KUKA KRL program: EPS_2_25618_SANMH10_A_20250918115518.src

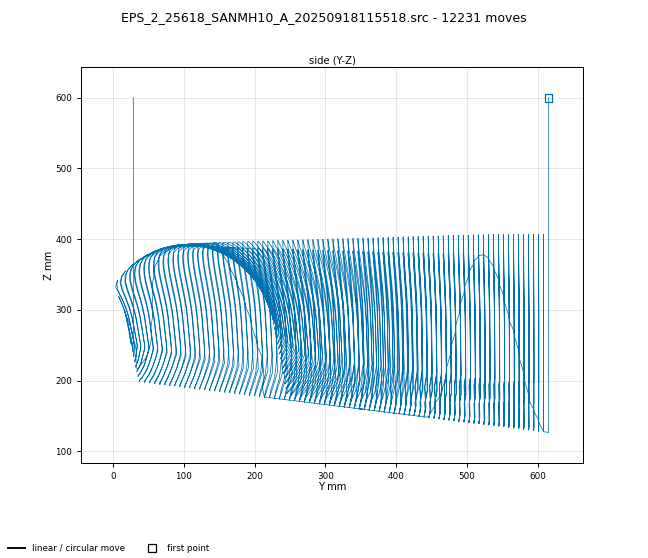
[picture p0: tool path of EPS_2_25618_SANMH10_A_20250918115518.src, 12231 of 12233 moves have a stored position in this frame; points joined in program order, loops and branches not executed]
&ACCESS RVP
&REL 4
&COMMENT QRS 19112012
&PARAM EDITMASK = *
DEF PART()
EXT BAS (BAS_COMMAND :IN,REAL :IN )
INT I
BAS (#INITMOV,0 )

;KUKA QRS Post kuka4.cps  Date:22-06-2017 !

File_ID=2846

QRS_PRE_INIT()

;Init var - Until changes are made in qrs_pre_init
Outlet_Square_prg=0
Inlet_1_Square_prg=0
Inlet_2_Square_prg=0
Inlet_3_Square_prg=0
Inlet_4_Square_prg=0
Inlet_5_Square_prg=0

Outlet_1={X 0.000, Y 546.330, Z 306.500, B 0.000, E1 0.000 }
Inlet_1={X 0.000, Y 548.460, Z 276.500, B 0.000, E1 118.000 }
Outlet_1_type=201
Inlet_1_type=201
;QRS#1=Sidecore dimensions
;QRS#2=200-8" PVC SDR 35
;QRS#3=200-8" PVC SDR 35
;QRS#4=
;QRS#5=
;QRS#6=
;QRS#7=
;QRS#8=
;QRS#9=12-08 PSX
;QRS#10=12-08 PSX
;QRS#11=
;QRS#12=
;QRS#13=
;QRS#14=
;QRS#15=
;QRS#16=1220x127x686 2,25'
;QRS#17=EPS Height
;QRS#18=407
;QRS#19=*
;QRS#20= UPDATED VERSION 22-06-2017
;QRS#21=*
Outlet_Square=0100
Inlet_1_Square=0100
Inlet_2_Square=0
Inlet_3_Square=0
Inlet_4_Square=0
Inlet_5_Square=0
Mill_Square=1
Outlet_Square_Prg=204
Inlet_1_Square_prg=204

QRS_INIT()

$ADVANCE=5

; T1
PTP {E1 173.646,E2 173.646}
PTP {X 0,Y 615.451,A -85,B 0,C 180,E1 173.646,E2 173.646,E3 0,E4 0,E5 0,E6 0}
QRS_SPEED_INIT()
LIN {X 0,Y 615.451,Z 600,A -85,B 0,C 180,E1 173.646,E2 173.646,E3 0,E4 0,E5 0,E6 0} C_VEL
LIN {X 0,Y 615.451,Z 136.872,A -85,B 0,C 180,E1 173.646,E2 173.646} C_VEL
LIN {X 0,Y 615.451,Z 128.693,A -85,B 0,C 180,E1 173.646,E2 173.646} C_VEL
LIN {X 0,Y 615.444,Z 126.693,A -85,B 0,C 180,E1 173.46,E2 173.46} C_VEL
LIN {X 0,Y 615.447,Z 126.714,A -85,B 0,C 180,E1 171.214,E2 171.214} C_VEL
LIN {X 0,Y 615.498,Z 142.353,A -85,B 0,C 180,E1 168.64,E2 168.64} C_VEL
LIN {X 0,Y 615.49,Z 160.105,A -85,B 0,C 180,E1 165.759,E2 165.759} C_VEL
LIN {X 0,Y 615.486,Z 165.964,A -85,B 0,C 180,E1 164.816,E2 164.816} C_VEL
LIN {X 0,Y 615.488,Z 273.613,A -85,B 0,C 180,E1 163.53,E2 163.53} C_VEL
LIN {X 0,Y 615.478,Z 286.482,A -85,B 0,C 180,E1 163.242,E2 163.242} C_VEL
LIN {X 0,Y 615.49,Z 299.343,A -85,B 0,C 180,E1 162.815,E2 162.815} C_VEL
LIN {X 0,Y 615.492,Z 310.759,A -85,B 0,C 180,E1 162.301,E2 162.301} C_VEL
LIN {X 0,Y 615.481,Z 322.204,A -85,B 0,C 180,E1 161.638,E2 161.638} C_VEL
LIN {X 0,Y 615.499,Z 333.228,A -85,B 0,C 180,E1 160.835,E2 160.835} C_VEL
LIN {X 0,Y 615.498,Z 342.752,A -85,B 0,C 180,E1 159.967,E2 159.967} C_VEL
LIN {X 0,Y 615.498,Z 350.589,A -85,B 0,C 180,E1 159.094,E2 159.094} C_VEL
LIN {X 0,Y 615.498,Z 358.274,A -85,B 0,C 180,E1 158.04,E2 158.04} C_VEL
LIN {X 0,Y 615.497,Z 363.428,A -85,B 0,C 180,E1 157.156,E2 157.156} C_VEL
LIN {X 0,Y 615.495,Z 368.74,A -85,B 0,C 180,E1 155.991,E2 155.991} C_VEL
LIN {X 0,Y 615.496,Z 372.068,A -85,B 0,C 180,E1 155.008,E2 155.008} C_VEL
LIN {X 0,Y 615.493,Z 373.871,A -85,B 0,C 180,E1 154.284,E2 154.284} C_VEL
LIN {X 0,Y 615.498,Z 375.211,A -85,B 0,C 180,E1 153.556,E2 153.556} C_VEL
LIN {X 0,Y 615.493,Z 376.024,A -85,B 0,C 180,E1 152.823,E2 152.823} C_VEL
LIN {X 0,Y 615.498,Z 376.298,A -85,B 0,C 180,E1 151.549,E2 151.549} C_VEL
LIN {X 0,Y 615.497,Z 374.962,A -85,B 0,C 180,E1 150.205,E2 150.205} C_VEL
LIN {X 0,Y 615.495,Z 372.101,A -85,B 0,C 180,E1 148.914,E2 148.914} C_VEL
LIN {X 0,Y 615.494,Z 369.013,A -85,B 0,C 180,E1 147.992,E2 147.992} C_VEL
LIN {X 0,Y 615.496,Z 363.479,A -85,B 0,C 180,E1 146.764,E2 146.764} C_VEL
LIN {X 0,Y 615.496,Z 356.718,A -85,B 0,C 180,E1 145.639,E2 145.639} C_VEL
LIN {X 0,Y 615.495,Z 348.697,A -85,B 0,C 180,E1 144.585,E2 144.585} C_VEL
LIN {X 0,Y 615.495,Z 340.536,A -85,B 0,C 180,E1 143.723,E2 143.723} C_VEL
LIN {X 0,Y 615.498,Z 331.142,A -85,B 0,C 180,E1 142.911,E2 142.911} C_VEL
LIN {X 0,Y 615.464,Z 320.86,A -85,B 0,C 180,E1 142.184,E2 142.184} C_VEL
LIN {X 0,Y 615.468,Z 309.903,A -85,B 0,C 180,E1 141.565,E2 141.565} C_VEL
LIN {X 0,Y 615.497,Z 297.229,A -85,B 0,C 180,E1 141.017,E2 141.017} C_VEL
LIN {X 0,Y 615.49,Z 285.344,A -85,B 0,C 180,E1 140.637,E2 140.637} C_VEL
LIN {X 0,Y 615.494,Z 272.35,A -85,B 0,C 180,E1 140.358,E2 140.358} C_VEL
LIN {X 0,Y 615.497,Z 165.933,A -85,B 0,C 180,E1 139.09,E2 139.09} C_VEL
LIN {X 0,Y 615.494,Z 148.019,A -85,B 0,C 180,E1 136.193,E2 136.193} C_VEL
LIN {X 0,Y 615.499,Z 130.019,A -85,B 0,C 180,E1 133.244,E2 133.244} C_VEL
LIN {X 0,Y 615.452,Z 126.693,A -85,B 0,C 180,E1 132.659,E2 132.659} C_VEL
LIN {X 0,Y 615.434,Z 126.696,A -85,B 0,C 180,E1 130.082,E2 130.082} C_VEL
LIN {X 0,Y 615.438,Z 126.697,A -85,B 0,C 180,E1 128.005,E2 128.005} C_VEL
LIN {X 0,Y 615.477,Z 126.699,A -85,B 0,C 180,E1 125.617,E2 125.617} C_VEL
LIN {X 0,Y 615.485,Z 126.694,A -85,B 0,C 180,E1 123.237,E2 123.237} C_VEL
LIN {X 0,Y 615.452,Z 126.693,A -85,B 0,C 180,E1 120.922,E2 120.922} C_VEL
LIN {X 0,Y 615.431,Z 126.696,A -85,B 0,C 180,E1 118.44,E2 118.44} C_VEL
LIN {X 0,Y 615.498,Z 126.697,A -85,B 0,C 180,E1 115.57,E2 115.57} C_VEL
LIN {X 0,Y 615.435,Z 126.695,A -85,B 0,C 180,E1 112.847,E2 112.847} C_VEL
LIN {X 0,Y 615.431,Z 126.697,A -85,B 0,C 180,E1 110.541,E2 110.541} C_VEL
LIN {X 0,Y 615.48,Z 126.699,A -85,B 0,C 180,E1 107.958,E2 107.958} C_VEL
LIN {X 0,Y 615.448,Z 126.694,A -85,B 0,C 180,E1 105.228,E2 105.228} C_VEL
LIN {X 0,Y 615.443,Z 126.694,A -85,B 0,C 180,E1 103.203,E2 103.203} C_VEL
LIN {X 0,Y 615.428,Z 126.696,A -85,B 0,C 180,E1 100.857,E2 100.857} C_VEL
LIN {X 0,Y 615.439,Z 126.698,A -85,B 0,C 180,E1 98.538,E2 98.538} C_VEL
LIN {X 0,Y 615.499,Z 126.694,A -85,B 0,C 180,E1 95.899,E2 95.899} C_VEL
LIN {X 0,Y 615.433,Z 126.695,A -85,B 0,C 180,E1 93.274,E2 93.274} C_VEL
LIN {X 0,Y 615.432,Z 126.696,A -85,B 0,C 180,E1 91.309,E2 91.309} C_VEL
LIN {X 0,Y 615.432,Z 126.696,A -85,B 0,C 180,E1 89.346,E2 89.346} C_VEL
LIN {X 0,Y 615.432,Z 126.696,A -85,B 0,C 180,E1 87.382,E2 87.382} C_VEL
LIN {X 0,Y 615.431,Z 126.696,A -85,B 0,C 180,E1 85.416,E2 85.416} C_VEL
LIN {X 0,Y 615.43,Z 126.696,A -85,B 0,C 180,E1 83.443,E2 83.443} C_VEL
LIN {X 0,Y 615.429,Z 126.696,A -85,B 0,C 180,E1 81.463,E2 81.463} C_VEL
LIN {X 0,Y 615.429,Z 126.697,A -85,B 0,C 180,E1 79.143,E2 79.143} C_VEL
LIN {X 0,Y 615.454,Z 126.699,A -85,B 0,C 180,E1 76.799,E2 76.799} C_VEL
LIN {X 0,Y 615.464,Z 126.695,A -85,B 0,C 180,E1 74.095,E2 74.095} C_VEL
LIN {X 0,Y 615.425,Z 126.697,A -85,B 0,C 180,E1 71.414,E2 71.414} C_VEL
LIN {X 0,Y 615.497,Z 126.698,A -85,B 0,C 180,E1 68.569,E2 68.569} C_VEL
LIN {X 0,Y 615.425,Z 126.697,A -85,B 0,C 180,E1 65.726,E2 65.726} C_VEL
LIN {X 0,Y 615.425,Z 126.697,A -85,B 0,C 180,E1 63.554,E2 63.554} C_VEL
LIN {X 0,Y 615.482,Z 126.697,A -85,B 0,C 180,E1 60.594,E2 60.594} C_VEL
LIN {X 0,Y 615.449,Z 126.696,A -85,B 0,C 180,E1 58.313,E2 58.313} C_VEL
LIN {X 0,Y 615.425,Z 126.697,A -85,B 0,C 180,E1 55.975,E2 55.975} C_VEL
LIN {X 0,Y 615.484,Z 126.7,A -85,B 0,C 180,E1 53.065,E2 53.065} C_VEL
LIN {X 0,Y 615.428,Z 126.697,A -85,B 0,C 180,E1 50.246,E2 50.246} C_VEL
LIN {X 0,Y 615.421,Z 126.698,A -85,B 0,C 180,E1 47.927,E2 47.927} C_VEL
LIN {X 0,Y 615.425,Z 126.698,A -85,B 0,C 180,E1 45.846,E2 45.846} C_VEL
LIN {X 0,Y 615.487,Z 126.7,A -85,B 0,C 180,E1 43.245,E2 43.245} C_VEL
LIN {X 0,Y 615.44,Z 126.697,A -85,B 0,C 180,E1 40.611,E2 40.611} C_VEL
LIN {X 0,Y 615.467,Z 126.696,A -85,B 0,C 180,E1 38.906,E2 38.906} C_VEL
LIN {X 0,Y 615.424,Z 126.697,A -85,B 0,C 180,E1 36.43,E2 36.43} C_VEL
LIN {X 0,Y 615.471,Z 126.701,A -85,B 0,C 180,E1 33.533,E2 33.533} C_VEL
LIN {X 0,Y 615.448,Z 126.697,A -85,B 0,C 180,E1 30.922,E2 30.922} C_VEL
LIN {X 0,Y 615.42,Z 126.698,A -85,B 0,C 180,E1 28.44,E2 28.44} C_VEL
LIN {X 0,Y 615.471,Z 126.7,A -85,B 0,C 180,E1 25.717,E2 25.717} C_VEL
LIN {X 0,Y 615.428,Z 126.698,A -85,B 0,C 180,E1 22.847,E2 22.847} C_VEL
LIN {X 0,Y 615.419,Z 126.698,A -85,B 0,C 180,E1 20.542,E2 20.542} C_VEL
LIN {X 0,Y 615.461,Z 126.7,A -85,B 0,C 180,E1 17.958,E2 17.958} C_VEL
LIN {X 0,Y 615.443,Z 126.698,A -85,B 0,C 180,E1 15.227,E2 15.227} C_VEL
LIN {X 0,Y 615.437,Z 126.698,A -85,B 0,C 180,E1 13.203,E2 13.203} C_VEL
LIN {X 0,Y 615.417,Z 126.699,A -85,B 0,C 180,E1 10.858,E2 10.858} C_VEL
LIN {X 0,Y 615.426,Z 126.699,A -85,B 0,C 180,E1 8.538,E2 8.538} C_VEL
LIN {X 0,Y 615.498,Z 126.699,A -85,B 0,C 180,E1 5.899,E2 5.899} C_VEL
LIN {X 0,Y 615.425,Z 126.698,A -85,B 0,C 180,E1 3.273,E2 3.273} C_VEL
LIN {X 0,Y 615.424,Z 126.699,A -85,B 0,C 180,E1 1.309,E2 1.309} C_VEL
LIN {X 0,Y 615.424,Z 126.698,A -85,B 0,C 180,E1 -0.654,E2 -0.654} C_VEL
LIN {X 0,Y 615.424,Z 126.699,A -85,B 0,C 180,E1 -2.618,E2 -2.618} C_VEL
LIN {X 0,Y 615.423,Z 126.699,A -85,B 0,C 180,E1 -4.585,E2 -4.585} C_VEL
LIN {X 0,Y 615.422,Z 126.699,A -85,B 0,C 180,E1 -6.557,E2 -6.557} C_VEL
LIN {X 0,Y 615.421,Z 126.699,A -85,B 0,C 180,E1 -8.537,E2 -8.537} C_VEL
LIN {X 0,Y 615.416,Z 126.699,A -85,B 0,C 180,E1 -10.858,E2 -10.858} C_VEL
LIN {X 0,Y 615.438,Z 126.7,A -85,B 0,C 180,E1 -13.202,E2 -13.202} C_VEL
LIN {X 0,Y 615.461,Z 126.699,A -85,B 0,C 180,E1 -15.906,E2 -15.906} C_VEL
LIN {X 0,Y 615.414,Z 126.7,A -85,B 0,C 180,E1 -18.648,E2 -18.648} C_VEL
LIN {X 0,Y 615.49,Z 126.7,A -85,B 0,C 180,E1 -21.432,E2 -21.432} C_VEL
LIN {X 0,Y 615.416,Z 126.699,A -85,B 0,C 180,E1 -24.275,E2 -24.275} C_VEL
LIN {X 0,Y 615.413,Z 126.7,A -85,B 0,C 180,E1 -26.448,E2 -26.448} C_VEL
LIN {X 0,Y 615.477,Z 126.702,A -85,B 0,C 180,E1 -29.407,E2 -29.407} C_VEL
LIN {X 0,Y 615.445,Z 126.7,A -85,B 0,C 180,E1 -31.688,E2 -31.688} C_VEL
LIN {X 0,Y 615.416,Z 126.7,A -85,B 0,C 180,E1 -34.027,E2 -34.027} C_VEL
LIN {X 0,Y 615.463,Z 126.7,A -85,B 0,C 180,E1 -36.935,E2 -36.935} C_VEL
LIN {X 0,Y 615.423,Z 126.7,A -85,B 0,C 180,E1 -39.755,E2 -39.755} C_VEL
LIN {X 0,Y 615.411,Z 126.7,A -85,B 0,C 180,E1 -42.073,E2 -42.073} C_VEL
LIN {X 0,Y 615.413,Z 126.7,A -85,B 0,C 180,E1 -44.156,E2 -44.156} C_VEL
LIN {X 0,Y 615.412,Z 126.7,A -85,B 0,C 180,E1 -46.01,E2 -46.01} C_VEL
LIN {X 0,Y 615.444,Z 126.7,A -85,B 0,C 180,E1 -48.524,E2 -48.524} C_VEL
LIN {X 0,Y 615.466,Z 126.7,A -85,B 0,C 180,E1 -51.095,E2 -51.095} C_VEL
LIN {X 0,Y 615.417,Z 126.7,A -85,B 0,C 180,E1 -53.571,E2 -53.571} C_VEL
LIN {X 0,Y 615.459,Z 126.699,A -85,B 0,C 180,E1 -56.47,E2 -56.47} C_VEL
LIN {X 0,Y 615.448,Z 126.7,A -85,B 0,C 180,E1 -59.079,E2 -59.079} C_VEL
LIN {X 0,Y 615.414,Z 126.699,A -85,B 0,C 180,E1 -61.563,E2 -61.563} C_VEL
LIN {X 0,Y 615.414,Z 126.699,A -85,B 0,C 180,E1 -63.553,E2 -63.553} C_VEL
LIN {X 0,Y 615.433,Z 126.699,A -85,B 0,C 180,E1 -66.004,E2 -66.004} C_VEL
LIN {X 0,Y 615.424,Z 126.78,A -85,B 0,C 180,E1 -67.838,E2 -67.838} C_VEL
LIN {X 0,Y 615.496,Z 145.823,A -85,B 0,C 180,E1 -70.49,E2 -70.49} C_VEL
LIN {X 0,Y 615.458,Z 165.936,A -85,B 0,C 180,E1 -73.242,E2 -73.242} C_VEL
LIN {X 0,Y 615.475,Z 185.711,A -85,B 0,C 180,E1 -75.916,E2 -75.916} C_VEL
LIN {X 0,Y 615.46,Z 194.649,A -85,B 0,C 180,E1 -77.114,E2 -77.114} C_VEL
LIN {X 0,Y 615.488,Z 302.864,A -85,B 0,C 180,E1 -78.411,E2 -78.411} C_VEL
LIN {X 0,Y 615.477,Z 315.368,A -85,B 0,C 180,E1 -78.682,E2 -78.682} C_VEL
LIN {X 0,Y 615.488,Z 328.616,A -85,B 0,C 180,E1 -79.113,E2 -79.113} C_VEL
LIN {X 0,Y 615.477,Z 340.49,A -85,B 0,C 180,E1 -79.64,E2 -79.64} C_VEL
LIN {X 0,Y 615.494,Z 352.003,A -85,B 0,C 180,E1 -80.305,E2 -80.305} C_VEL
LIN {X 0,Y 615.499,Z 362.349,A -85,B 0,C 180,E1 -81.05,E2 -81.05} C_VEL
LIN {X 0,Y 615.497,Z 370.818,A -85,B 0,C 180,E1 -81.795,E2 -81.795} C_VEL
LIN {X 0,Y 615.498,Z 378.611,A -85,B 0,C 180,E1 -82.62,E2 -82.62} C_VEL
LIN {X 0,Y 615.496,Z 386.207,A -85,B 0,C 180,E1 -83.609,E2 -83.609} C_VEL
LIN {X 0,Y 615.498,Z 393.208,A -85,B 0,C 180,E1 -84.759,E2 -84.759} C_VEL
LIN {X 0,Y 615.494,Z 397.854,A -85,B 0,C 180,E1 -85.744,E2 -85.744} C_VEL
LIN {X 0,Y 615.494,Z 401.401,A -85,B 0,C 180,E1 -86.728,E2 -86.728} C_VEL
LIN {X 0,Y 615.497,Z 403.234,A -85,B 0,C 180,E1 -87.383,E2 -87.383} C_VEL
LIN {X 0,Y 615.5,Z 404.608,A -85,B 0,C 180,E1 -88.038,E2 -88.038} C_VEL
LIN {X 0,Y 615.496,Z 406.174,A -85,B 0,C 180,E1 -89.346,E2 -89.346} C_VEL
LIN {X 0,Y 615.494,Z 406.389,A -85,B 0,C 180,E1 -90.001,E2 -90.001} C_VEL
LIN {X 0,Y 615.495,Z 405.579,A -85,B 0,C 180,E1 -91.309,E2 -91.309} C_VEL
LIN {X 0,Y 615.5,Z 404.607,A -85,B 0,C 180,E1 -91.964,E2 -91.964} C_VEL
LIN {X 0,Y 615.497,Z 403.232,A -85,B 0,C 180,E1 -92.618,E2 -92.618} C_VEL
LIN {X 0,Y 615.496,Z 400.348,A -85,B 0,C 180,E1 -93.601,E2 -93.601} C_VEL
LIN {X 0,Y 615.498,Z 396.439,A -85,B 0,C 180,E1 -94.585,E2 -94.585} C_VEL
LIN {X 0,Y 615.499,Z 391.402,A -85,B 0,C 180,E1 -95.57,E2 -95.57} C_VEL
LIN {X 0,Y 615.497,Z 384.869,A -85,B 0,C 180,E1 -96.583,E2 -96.583} C_VEL
LIN {X 0,Y 615.497,Z 377.128,A -85,B 0,C 180,E1 -97.546,E2 -97.546} C_VEL
LIN {X 0,Y 615.498,Z 369.039,A -85,B 0,C 180,E1 -98.372,E2 -98.372} C_VEL
LIN {X 0,Y 615.499,Z 359.16,A -85,B 0,C 180,E1 -99.199,E2 -99.199} C_VEL
LIN {X 0,Y 615.488,Z 347.972,A -85,B 0,C 180,E1 -99.946,E2 -99.946} C_VEL
LIN {X 0,Y 615.482,Z 337.012,A -85,B 0,C 180,E1 -100.528,E2 -100.528} C_VEL
LIN {X 0,Y 615.48,Z 324.482,A -85,B 0,C 180,E1 -101.04,E2 -101.04} C_VEL
LIN {X 0,Y 615.479,Z 312.044,A -85,B 0,C 180,E1 -101.402,E2 -101.402} C_VEL
LIN {X 0,Y 615.493,Z 298.427,A -85,B 0,C 180,E1 -101.652,E2 -101.652} C_VEL
LIN {X 0,Y 615.46,Z 194.641,A -85,B 0,C 180,E1 -102.888,E2 -102.888} C_VEL
LIN {X 0,Y 615.497,Z 173.46,A -85,B 0,C 180,E1 -105.735,E2 -105.735} C_VEL
LIN {X 0,Y 615.482,Z 152.104,A -85,B 0,C 180,E1 -108.647,E2 -108.647} C_VEL
LIN {X 0,Y 615.494,Z 131.977,A -85,B 0,C 180,E1 -111.432,E2 -111.432} C_VEL
LIN {X 0,Y 615.423,Z 126.699,A -85,B 0,C 180,E1 -112.187,E2 -112.187} C_VEL
LIN {X 0,Y 615.418,Z 126.699,A -85,B 0,C 180,E1 -114.275,E2 -114.275} C_VEL
LIN {X 0,Y 615.418,Z 126.699,A -85,B 0,C 180,E1 -116.448,E2 -116.448} C_VEL
LIN {X 0,Y 615.479,Z 126.7,A -85,B 0,C 180,E1 -119.407,E2 -119.407} C_VEL
LIN {X 0,Y 615.448,Z 126.697,A -85,B 0,C 180,E1 -121.688,E2 -121.688} C_VEL
LIN {X 0,Y 615.422,Z 126.698,A -85,B 0,C 180,E1 -124.027,E2 -124.027} C_VEL
LIN {X 0,Y 615.48,Z 126.7,A -85,B 0,C 180,E1 -126.935,E2 -126.935} C_VEL
LIN {X 0,Y 615.428,Z 126.697,A -85,B 0,C 180,E1 -129.755,E2 -129.755} C_VEL
LIN {X 0,Y 615.424,Z 126.698,A -85,B 0,C 180,E1 -132.073,E2 -132.073} C_VEL
LIN {X 0,Y 615.428,Z 126.698,A -85,B 0,C 180,E1 -134.155,E2 -134.155} C_VEL
LIN {X 0,Y 615.493,Z 126.7,A -85,B 0,C 180,E1 -136.756,E2 -136.756} C_VEL
LIN {X 0,Y 615.442,Z 126.695,A -85,B 0,C 180,E1 -139.39,E2 -139.39} C_VEL
LIN {X 0,Y 615.43,Z 126.697,A -85,B 0,C 180,E1 -141.927,E2 -141.927} C_VEL
LIN {X 0,Y 615.47,Z 126.699,A -85,B 0,C 180,E1 -144.383,E2 -144.383} C_VEL
LIN {X 0,Y 615.485,Z 126.695,A -85,B 0,C 180,E1 -146.764,E2 -146.764} C_VEL
LIN {X 0,Y 615.452,Z 126.694,A -85,B 0,C 180,E1 -149.078,E2 -149.078} C_VEL
LIN {X 0,Y 615.431,Z 126.696,A -85,B 0,C 180,E1 -151.56,E2 -151.56} C_VEL
LIN {X 0,Y 615.498,Z 126.697,A -85,B 0,C 180,E1 -154.43,E2 -154.43} C_VEL
LIN {X 0,Y 615.437,Z 126.695,A -85,B 0,C 180,E1 -157.153,E2 -157.153} C_VEL
LIN {X 0,Y 615.435,Z 126.696,A -85,B 0,C 180,E1 -159.457,E2 -159.457} C_VEL
LIN {X 0,Y 615.489,Z 126.7,A -85,B 0,C 180,E1 -162.043,E2 -162.043} C_VEL
LIN {X 0,Y 615.451,Z 126.693,A -85,B 0,C 180,E1 -164.773,E2 -164.773} C_VEL
LIN {X 0,Y 615.447,Z 126.693,A -85,B 0,C 180,E1 -166.798,E2 -166.798} C_VEL
LIN {X 0,Y 615.437,Z 126.695,A -85,B 0,C 180,E1 -169.138,E2 -169.138} C_VEL
LIN {X 0,Y 615.455,Z 126.697,A -85,B 0,C 180,E1 -171.463,E2 -171.463} C_VEL
LIN {X 0,Y 615.499,Z 126.69,A -85,B 0,C 180,E1 -174.102,E2 -174.102} C_VEL
LIN {X 0,Y 615.442,Z 126.693,A -85,B 0,C 180,E1 -176.727,E2 -176.727} C_VEL
LIN {X 0,Y 615.442,Z 126.693,A -85,B 0,C 180,E1 -178.691,E2 -178.691} C_VEL
LIN {X 0,Y 615.466,Z 126.698,A -85,B 0,C 180,E1 -181.309,E2 -181.309} C_VEL
LIN {X 0,Y 615.486,Z 126.691,A -85,B 0,C 180,E1 -183.929,E2 -183.929} C_VEL
LIN {X 0,Y 615.444,Z 126.693,A -85,B 0,C 180,E1 -186.54,E2 -186.54} C_VEL
LIN {X 0,Y 614.772,Z 126.843,A -85,B 0,C 180,E1 -186.904,E2 -186.904} C_VEL
LIN {X 0,Y 611.949,Z 127.262,A -85,B 0,C 180,E1 -187.474,E2 -187.474} C_VEL
LIN {X 0,Y 609.112,Z 127.617,A -85,B 0,C 180,E1 -188.048,E2 -188.048} C_VEL
LIN {X 0,Y 608.43,Z 127.691,A -85,B 0,C 180,E1 -188.418,E2 -188.418} C_VEL
LIN {X 0,Y 608.425,Z 127.751,A -85,B 0,C 180,E1 -188.72,E2 -188.72} C_VEL
LIN {X 0,Y 608.481,Z 141.815,A -85,B 0,C 180,E1 -191.058,E2 -191.058} C_VEL
LIN {X 0,Y 608.474,Z 159.127,A -85,B 0,C 180,E1 -193.894,E2 -193.894} C_VEL
LIN {X 0,Y 608.461,Z 166.295,A -85,B 0,C 180,E1 -195.042,E2 -195.042} C_VEL
LIN {X 0,Y 608.556,Z 273.083,A -85,B 0,C 180,E1 -196.324,E2 -196.324} C_VEL
LIN {X 0,Y 608.524,Z 286.825,A -85,B 0,C 180,E1 -196.633,E2 -196.633} C_VEL
LIN {X 0,Y 608.524,Z 298.998,A -85,B 0,C 180,E1 -197.042,E2 -197.042} C_VEL
LIN {X 0,Y 608.52,Z 310.581,A -85,B 0,C 180,E1 -197.562,E2 -197.562} C_VEL
LIN {X 0,Y 608.478,Z 322.455,A -85,B 0,C 180,E1 -198.253,E2 -198.253} C_VEL
LIN {X 0,Y 608.471,Z 333.275,A -85,B 0,C 180,E1 -199.044,E2 -199.044} C_VEL
LIN {X 0,Y 608.467,Z 342.896,A -85,B 0,C 180,E1 -199.922,E2 -199.922} C_VEL
LIN {X 0,Y 608.456,Z 350.516,A -85,B 0,C 180,E1 -200.768,E2 -200.768} C_VEL
LIN {X 0,Y 608.456,Z 358.581,A -85,B 0,C 180,E1 -201.87,E2 -201.87} C_VEL
LIN {X 0,Y 608.447,Z 363.797,A -85,B 0,C 180,E1 -202.765,E2 -202.765} C_VEL
LIN {X 0,Y 608.441,Z 368.826,A -85,B 0,C 180,E1 -203.846,E2 -203.846} C_VEL
LIN {X 0,Y 608.433,Z 372.58,A -85,B 0,C 180,E1 -204.937,E2 -204.937} C_VEL
LIN {X 0,Y 608.427,Z 375.165,A -85,B 0,C 180,E1 -206.037,E2 -206.037} C_VEL
LIN {X 0,Y 608.435,Z 376.654,A -85,B 0,C 180,E1 -207.198,E2 -207.198} C_VEL
LIN {X 0,Y 608.423,Z 376.851,A -85,B 0,C 180,E1 -208.611,E2 -208.611} C_VEL
LIN {X 0,Y 608.422,Z 375.314,A -85,B 0,C 180,E1 -209.963,E2 -209.963} C_VEL
LIN {X 0,Y 608.442,Z 374.141,A -85,B 0,C 180,E1 -210.547,E2 -210.547} C_VEL
LIN {X 0,Y 608.429,Z 370.828,A -85,B 0,C 180,E1 -211.707,E2 -211.707} C_VEL
LIN {X 0,Y 608.447,Z 366.018,A -85,B 0,C 180,E1 -212.881,E2 -212.881} C_VEL
LIN {X 0,Y 608.441,Z 359.505,A -85,B 0,C 180,E1 -214.072,E2 -214.072} C_VEL
LIN {X 0,Y 608.467,Z 352.616,A -85,B 0,C 180,E1 -215.062,E2 -215.062} C_VEL
LIN {X 0,Y 608.46,Z 343.639,A -85,B 0,C 180,E1 -216.092,E2 -216.092} C_VEL
LIN {X 0,Y 608.492,Z 333.766,A -85,B 0,C 180,E1 -217.005,E2 -217.005} C_VEL
LIN {X 0,Y 608.463,Z 323.824,A -85,B 0,C 180,E1 -217.747,E2 -217.747} C_VEL
LIN {X 0,Y 608.471,Z 313.346,A -85,B 0,C 180,E1 -218.381,E2 -218.381} C_VEL
LIN {X 0,Y 608.506,Z 301.271,A -85,B 0,C 180,E1 -218.957,E2 -218.957} C_VEL
LIN {X 0,Y 608.551,Z 288.756,A -85,B 0,C 180,E1 -219.402,E2 -219.402} C_VEL
LIN {X 0,Y 608.537,Z 275.769,A -85,B 0,C 180,E1 -219.717,E2 -219.717} C_VEL
LIN {X 0,Y 608.552,Z 255.918,A -85,B 0,C 180,E1 -219.985,E2 -219.985} C_VEL
LIN {X 0,Y 608.47,Z 166.173,A -85,B 0,C 180,E1 -221.053,E2 -221.053} C_VEL
LIN {X 0,Y 608.478,Z 148.886,A -85,B 0,C 180,E1 -223.869,E2 -223.869} C_VEL
LIN {X 0,Y 608.507,Z 131.819,A -85,B 0,C 180,E1 -226.688,E2 -226.688} C_VEL
LIN {X 0,Y 608.437,Z 127.691,A -85,B 0,C 180,E1 -227.386,E2 -227.386} C_VEL
LIN {X 0,Y 608.422,Z 127.691,A -85,B 0,C 180,E1 -229.694,E2 -229.694} C_VEL
LIN {X 0,Y 608.444,Z 127.693,A -85,B 0,C 180,E1 -232.251,E2 -232.251} C_VEL
LIN {X 0,Y 608.42,Z 127.694,A -85,B 0,C 180,E1 -235.099,E2 -235.099} C_VEL
LIN {X 0,Y 608.417,Z 127.692,A -85,B 0,C 180,E1 -237.485,E2 -237.485} C_VEL
LIN {X 0,Y 608.454,Z 127.694,A -85,B 0,C 180,E1 -240.219,E2 -240.219} C_VEL
LIN {X 0,Y 608.406,Z 127.693,A -85,B 0,C 180,E1 -243.223,E2 -243.223} C_VEL
LIN {X 0,Y 608.417,Z 127.692,A -85,B 0,C 180,E1 -245.427,E2 -245.427} C_VEL
LIN {X 0,Y 608.457,Z 127.697,A -85,B 0,C 180,E1 -248.308,E2 -248.308} C_VEL
LIN {X 0,Y 608.418,Z 127.692,A -85,B 0,C 180,E1 -251.3,E2 -251.3} C_VEL
LIN {X 0,Y 608.442,Z 127.695,A -85,B 0,C 180,E1 -253.905,E2 -253.905} C_VEL
LIN {X 0,Y 608.436,Z 127.692,A -85,B 0,C 180,E1 -256.642,E2 -256.642} C_VEL
LIN {X 0,Y 608.417,Z 127.693,A -85,B 0,C 180,E1 -259.349,E2 -259.349} C_VEL
LIN {X 0,Y 608.476,Z 127.694,A -85,B 0,C 180,E1 -262.033,E2 -262.033} C_VEL
LIN {X 0,Y 608.421,Z 127.692,A -85,B 0,C 180,E1 -264.697,E2 -264.697} C_VEL
LIN {X 0,Y 608.438,Z 127.692,A -85,B 0,C 180,E1 -267.351,E2 -267.351} C_VEL
LIN {X 0,Y 608.478,Z 127.692,A -85,B 0,C 180,E1 -269.999,E2 -269.999} C_VEL
LIN {X 0,Y 608.428,Z 127.691,A -85,B 0,C 180,E1 -272.648,E2 -272.648} C_VEL
LIN {X 0,Y 608.431,Z 127.694,A -85,B 0,C 180,E1 -275.302,E2 -275.302} C_VEL
LIN {X 0,Y 608.469,Z 127.69,A -85,B 0,C 180,E1 -277.966,E2 -277.966} C_VEL
LIN {X 0,Y 608.41,Z 127.693,A -85,B 0,C 180,E1 -280.65,E2 -280.65} C_VEL
LIN {X 0,Y 608.438,Z 127.697,A -85,B 0,C 180,E1 -283.356,E2 -283.356} C_VEL
LIN {X 0,Y 608.427,Z 127.692,A -85,B 0,C 180,E1 -286.094,E2 -286.094} C_VEL
LIN {X 0,Y 608.432,Z 127.692,A -85,B 0,C 180,E1 -288.87,E2 -288.87} C_VEL
LIN {X 0,Y 608.456,Z 127.692,A -85,B 0,C 180,E1 -291.691,E2 -291.691} C_VEL
LIN {X 0,Y 608.415,Z 127.693,A -85,B 0,C 180,E1 -294.572,E2 -294.572} C_VEL
LIN {X 0,Y 608.473,Z 127.695,A -85,B 0,C 180,E1 -297.205,E2 -297.205} C_VEL
LIN {X 0,Y 608.407,Z 127.694,A -85,B 0,C 180,E1 -299.961,E2 -299.961} C_VEL
LIN {X 0,Y 608.414,Z 127.694,A -85,B 0,C 180,E1 -302.514,E2 -302.514} C_VEL
LIN {X 0,Y 608.423,Z 127.699,A -85,B 0,C 180,E1 -304.901,E2 -304.901} C_VEL
LIN {X 0,Y 608.43,Z 127.691,A -85,B 0,C 180,E1 -307.748,E2 -307.748} C_VEL
LIN {X 0,Y 608.4,Z 127.695,A -85,B 0,C 180,E1 -310.323,E2 -310.323} C_VEL
LIN {X 0,Y 608.447,Z 127.698,A -85,B 0,C 180,E1 -312.959,E2 -312.959} C_VEL
LIN {X 0,Y 608.404,Z 127.694,A -85,B 0,C 180,E1 -315.74,E2 -315.74} C_VEL
LIN {X 0,Y 608.406,Z 127.693,A -85,B 0,C 180,E1 -317.933,E2 -317.933} C_VEL
LIN {X 0,Y 608.434,Z 127.7,A -85,B 0,C 180,E1 -320.706,E2 -320.706} C_VEL
LIN {X 0,Y 608.433,Z 127.694,A -85,B 0,C 180,E1 -323.083,E2 -323.083} C_VEL
LIN {X 0,Y 608.42,Z 127.692,A -85,B 0,C 180,E1 -325.527,E2 -325.527} C_VEL
LIN {X 0,Y 608.418,Z 127.693,A -85,B 0,C 180,E1 -327.902,E2 -327.902} C_VEL
LIN {X 0,Y 608.437,Z 127.694,A -85,B 0,C 180,E1 -330.218,E2 -330.218} C_VEL
LIN {X 0,Y 608.398,Z 127.695,A -85,B 0,C 180,E1 -333.223,E2 -333.223} C_VEL
LIN {X 0,Y 608.407,Z 127.693,A -85,B 0,C 180,E1 -335.427,E2 -335.427} C_VEL
LIN {X 0,Y 608.45,Z 127.697,A -85,B 0,C 180,E1 -338.307,E2 -338.307} C_VEL
LIN {X 0,Y 608.406,Z 127.693,A -85,B 0,C 180,E1 -341.3,E2 -341.3} C_VEL
LIN {X 0,Y 608.428,Z 127.695,A -85,B 0,C 180,E1 -343.905,E2 -343.905} C_VEL
LIN {X 0,Y 608.427,Z 127.694,A -85,B 0,C 180,E1 -346.643,E2 -346.643} C_VEL
LIN {X 0,Y 608.402,Z 127.694,A -85,B 0,C 180,E1 -349.349,E2 -349.349} C_VEL
LIN {X 0,Y 608.464,Z 127.695,A -85,B 0,C 180,E1 -352.033,E2 -352.033} C_VEL
LIN {X 0,Y 608.413,Z 127.694,A -85,B 0,C 180,E1 -354.697,E2 -354.697} C_VEL
LIN {X 0,Y 608.423,Z 127.692,A -85,B 0,C 180,E1 -357.352,E2 -357.352} C_VEL
LIN {X 0,Y 608.469,Z 127.695,A -85,B 0,C 180,E1 -360,E2 -360} C_VEL
LIN {X 0,Y 608.419,Z 127.692,A -85,B 0,C 180,E1 -362.648,E2 -362.648} C_VEL
LIN {X 0,Y 608.417,Z 127.694,A -85,B 0,C 180,E1 -365.302,E2 -365.302} C_VEL
LIN {X 0,Y 608.461,Z 127.694,A -85,B 0,C 180,E1 -367.967,E2 -367.967} C_VEL
LIN {X 0,Y 608.4,Z 127.694,A -85,B 0,C 180,E1 -370.651,E2 -370.651} C_VEL
LIN {X 0,Y 608.426,Z 127.696,A -85,B 0,C 180,E1 -373.357,E2 -373.357} C_VEL
LIN {X 0,Y 608.421,Z 127.694,A -85,B 0,C 180,E1 -376.095,E2 -376.095} C_VEL
LIN {X 0,Y 608.42,Z 127.693,A -85,B 0,C 180,E1 -378.871,E2 -378.871} C_VEL
LIN {X 0,Y 608.448,Z 127.695,A -85,B 0,C 180,E1 -381.692,E2 -381.692} C_VEL
LIN {X 0,Y 608.402,Z 127.694,A -85,B 0,C 180,E1 -384.573,E2 -384.573} C_VEL
LIN {X 0,Y 608.456,Z 127.695,A -85,B 0,C 180,E1 -387.205,E2 -387.205} C_VEL
LIN {X 0,Y 608.4,Z 127.695,A -85,B 0,C 180,E1 -389.962,E2 -389.962} C_VEL
LIN {X 0,Y 608.401,Z 127.694,A -85,B 0,C 180,E1 -392.515,E2 -392.515} C_VEL
LIN {X 0,Y 608.409,Z 127.698,A -85,B 0,C 180,E1 -394.901,E2 -394.901} C_VEL
LIN {X 0,Y 608.422,Z 127.693,A -85,B 0,C 180,E1 -397.75,E2 -397.75} C_VEL
LIN {X 0,Y 608.395,Z 127.695,A -85,B 0,C 180,E1 -400.324,E2 -400.324} C_VEL
LIN {X 0,Y 608.435,Z 127.699,A -85,B 0,C 180,E1 -402.962,E2 -402.962} C_VEL
LIN {X 0,Y 608.397,Z 127.695,A -85,B 0,C 180,E1 -405.742,E2 -405.742} C_VEL
LIN {X 0,Y 608.397,Z 127.694,A -85,B 0,C 180,E1 -407.934,E2 -407.934} C_VEL
LIN {X 0,Y 608.43,Z 127.698,A -85,B 0,C 180,E1 -410.707,E2 -410.707} C_VEL
LIN {X 0,Y 608.432,Z 127.696,A -85,B 0,C 180,E1 -413.084,E2 -413.084} C_VEL
LIN {X 0,Y 608.417,Z 127.693,A -85,B 0,C 180,E1 -415.528,E2 -415.528} C_VEL
LIN {X 0,Y 608.41,Z 127.693,A -85,B 0,C 180,E1 -417.903,E2 -417.903} C_VEL
LIN {X 0,Y 608.425,Z 127.694,A -85,B 0,C 180,E1 -420.219,E2 -420.219} C_VEL
LIN {X 0,Y 608.398,Z 127.696,A -85,B 0,C 180,E1 -423.224,E2 -423.224} C_VEL
LIN {X 0,Y 608.404,Z 127.694,A -85,B 0,C 180,E1 -425.428,E2 -425.428} C_VEL
LIN {X 0,Y 608.426,Z 127.895,A -85,B 0,C 180,E1 -427.728,E2 -427.728} C_VEL
LIN {X 0,Y 608.533,Z 142.063,A -85,B 0,C 180,E1 -429.729,E2 -429.729} C_VEL
LIN {X 0,Y 608.515,Z 160.953,A -85,B 0,C 180,E1 -432.352,E2 -432.352} C_VEL
LIN {X 0,Y 608.488,Z 182.361,A -85,B 0,C 180,E1 -435.28,E2 -435.28} C_VEL
LIN {X 0,Y 608.472,Z 195.196,A -85,B 0,C 180,E1 -436.984,E2 -436.984} C_VEL
LIN {X 0,Y 608.547,Z 302.981,A -85,B 0,C 180,E1 -438.277,E2 -438.277} C_VEL
LIN {X 0,Y 608.512,Z 316.239,A -85,B 0,C 180,E1 -438.572,E2 -438.572} C_VEL
LIN {X 0,Y 608.513,Z 328.16,A -85,B 0,C 180,E1 -438.965,E2 -438.965} C_VEL
LIN {X 0,Y 608.499,Z 340.646,A -85,B 0,C 180,E1 -439.52,E2 -439.52} C_VEL
LIN {X 0,Y 608.484,Z 352.207,A -85,B 0,C 180,E1 -440.192,E2 -440.192} C_VEL
LIN {X 0,Y 608.485,Z 362.602,A -85,B 0,C 180,E1 -440.946,E2 -440.946} C_VEL
LIN {X 0,Y 608.475,Z 371.118,A -85,B 0,C 180,E1 -441.699,E2 -441.699} C_VEL
LIN {X 0,Y 608.47,Z 378.965,A -85,B 0,C 180,E1 -442.534,E2 -442.534} C_VEL
LIN {X 0,Y 608.46,Z 386.289,A -85,B 0,C 180,E1 -443.485,E2 -443.485} C_VEL
LIN {X 0,Y 608.451,Z 391.869,A -85,B 0,C 180,E1 -444.366,E2 -444.366} C_VEL
LIN {X 0,Y 608.432,Z 396.953,A -85,B 0,C 180,E1 -445.363,E2 -445.363} C_VEL
LIN {X 0,Y 608.449,Z 400.898,A -85,B 0,C 180,E1 -446.358,E2 -446.358} C_VEL
LIN {X 0,Y 608.425,Z 403.811,A -85,B 0,C 180,E1 -447.352,E2 -447.352} C_VEL
LIN {X 0,Y 608.445,Z 405.202,A -85,B 0,C 180,E1 -448.015,E2 -448.015} C_VEL
LIN {X 0,Y 608.438,Z 406.784,A -85,B 0,C 180,E1 -449.339,E2 -449.339} C_VEL
LIN {X 0,Y 608.434,Z 407,A -85,B 0,C 180,E1 -450.001,E2 -450.001} C_VEL
LIN {X 0,Y 608.448,Z 406.183,A -85,B 0,C 180,E1 -451.324,E2 -451.324} C_VEL
LIN {X 0,Y 608.445,Z 405.2,A -85,B 0,C 180,E1 -451.986,E2 -451.986} C_VEL
LIN {X 0,Y 608.425,Z 403.808,A -85,B 0,C 180,E1 -452.649,E2 -452.649} C_VEL
LIN {X 0,Y 608.449,Z 400.894,A -85,B 0,C 180,E1 -453.643,E2 -453.643} C_VEL
LIN {X 0,Y 608.432,Z 396.948,A -85,B 0,C 180,E1 -454.638,E2 -454.638} C_VEL
LIN {X 0,Y 608.438,Z 390.873,A -85,B 0,C 180,E1 -455.801,E2 -455.801} C_VEL
LIN {X 0,Y 608.462,Z 384.231,A -85,B 0,C 180,E1 -456.8,E2 -456.8} C_VEL
LIN {X 0,Y 608.456,Z 375.984,A -85,B 0,C 180,E1 -457.801,E2 -457.801} C_VEL
LIN {X 0,Y 608.472,Z 367.53,A -85,B 0,C 180,E1 -458.636,E2 -458.636} C_VEL
LIN {X 0,Y 608.479,Z 357.084,A -85,B 0,C 180,E1 -459.474,E2 -459.474} C_VEL
LIN {X 0,Y 608.489,Z 346.747,A -85,B 0,C 180,E1 -460.145,E2 -460.145} C_VEL
LIN {X 0,Y 608.519,Z 335.258,A -85,B 0,C 180,E1 -460.74,E2 -460.74} C_VEL
LIN {X 0,Y 608.528,Z 322.877,A -85,B 0,C 180,E1 -461.225,E2 -461.225} C_VEL
LIN {X 0,Y 608.544,Z 309.415,A -85,B 0,C 180,E1 -461.597,E2 -461.597} C_VEL
LIN {X 0,Y 608.554,Z 297.043,A -85,B 0,C 180,E1 -461.808,E2 -461.808} C_VEL
LIN {X 0,Y 608.467,Z 195.098,A -85,B 0,C 180,E1 -463.017,E2 -463.017} C_VEL
LIN {X 0,Y 608.504,Z 174.797,A -85,B 0,C 180,E1 -465.749,E2 -465.749} C_VEL
LIN {X 0,Y 608.499,Z 154.811,A -85,B 0,C 180,E1 -468.497,E2 -468.497} C_VEL
LIN {X 0,Y 608.525,Z 137.017,A -85,B 0,C 180,E1 -470.98,E2 -470.98} C_VEL
LIN {X 0,Y 608.395,Z 127.697,A -85,B 0,C 180,E1 -472.319,E2 -472.319} C_VEL
LIN {X 0,Y 608.406,Z 127.694,A -85,B 0,C 180,E1 -474.574,E2 -474.574} C_VEL
LIN {X 0,Y 608.466,Z 127.695,A -85,B 0,C 180,E1 -477.204,E2 -477.204} C_VEL
LIN {X 0,Y 608.404,Z 127.695,A -85,B 0,C 180,E1 -479.961,E2 -479.961} C_VEL
LIN {X 0,Y 608.411,Z 127.694,A -85,B 0,C 180,E1 -482.515,E2 -482.515} C_VEL
LIN {X 0,Y 608.413,Z 127.7,A -85,B 0,C 180,E1 -485.28,E2 -485.28} C_VEL
LIN {X 0,Y 608.429,Z 127.691,A -85,B 0,C 180,E1 -487.75,E2 -487.75} C_VEL
LIN {X 0,Y 608.405,Z 127.695,A -85,B 0,C 180,E1 -490.324,E2 -490.324} C_VEL
LIN {X 0,Y 608.447,Z 127.698,A -85,B 0,C 180,E1 -492.961,E2 -492.961} C_VEL
LIN {X 0,Y 608.407,Z 127.693,A -85,B 0,C 180,E1 -495.741,E2 -495.741} C_VEL
LIN {X 0,Y 608.41,Z 127.693,A -85,B 0,C 180,E1 -497.934,E2 -497.934} C_VEL
LIN {X 0,Y 608.437,Z 127.7,A -85,B 0,C 180,E1 -500.707,E2 -500.707} C_VEL
LIN {X 0,Y 608.435,Z 127.693,A -85,B 0,C 180,E1 -503.084,E2 -503.084} C_VEL
LIN {X 0,Y 608.428,Z 127.691,A -85,B 0,C 180,E1 -505.528,E2 -505.528} C_VEL
LIN {X 0,Y 608.429,Z 127.692,A -85,B 0,C 180,E1 -507.903,E2 -507.903} C_VEL
LIN {X 0,Y 608.453,Z 127.694,A -85,B 0,C 180,E1 -510.22,E2 -510.22} C_VEL
LIN {X 0,Y 608.406,Z 127.693,A -85,B 0,C 180,E1 -513.224,E2 -513.224} C_VEL
LIN {X 0,Y 608.418,Z 127.692,A -85,B 0,C 180,E1 -515.427,E2 -515.427} C_VEL
LIN {X 0,Y 608.458,Z 127.696,A -85,B 0,C 180,E1 -518.308,E2 -518.308} C_VEL
LIN {X 0,Y 608.42,Z 127.692,A -85,B 0,C 180,E1 -521.299,E2 -521.299} C_VEL
LIN {X 0,Y 608.448,Z 127.696,A -85,B 0,C 180,E1 -523.906,E2 -523.906} C_VEL
LIN {X 0,Y 608.439,Z 127.691,A -85,B 0,C 180,E1 -526.643,E2 -526.643} C_VEL
LIN {X 0,Y 608.427,Z 127.693,A -85,B 0,C 180,E1 -529.35,E2 -529.35} C_VEL
LIN {X 0,Y 608.477,Z 127.692,A -85,B 0,C 180,E1 -532.033,E2 -532.033} C_VEL
LIN {X 0,Y 608.428,Z 127.691,A -85,B 0,C 180,E1 -534.698,E2 -534.698} C_VEL
LIN {X 0,Y 608.452,Z 127.692,A -85,B 0,C 180,E1 -537.352,E2 -537.352} C_VEL
LIN {X 0,Y 608.477,Z 127.689,A -85,B 0,C 180,E1 -540,E2 -540} C_VEL
LIN {X 0,Y 608.439,Z 127.689,A -85,B 0,C 180,E1 -542.648,E2 -542.648} C_VEL
LIN {X 0,Y 608.453,Z 127.695,A -85,B 0,C 180,E1 -545.302,E2 -545.302} C_VEL
LIN {X 0,Y 608.471,Z 127.688,A -85,B 0,C 180,E1 -547.967,E2 -547.967} C_VEL
LIN {X 0,Y 608.43,Z 127.691,A -85,B 0,C 180,E1 -548.418,E2 -548.418} C_VEL
LIN {X 0,Y 608.235,Z 128.2,A -85,B 0,C 180,E1 -548.696,E2 -548.696} C_VEL
LIN {X 0,Y 607.31,Z 130.36,A -85,B 0,C 180,E1 -549.12,E2 -549.12} C_VEL
LIN {X 0,Y 602.167,Z 139.623,A -85,B 0,C 180,E1 -550.495,E2 -550.495} C_VEL
LIN {X 0,Y 601.481,Z 142.55,A -85,B 0,C 180,E1 -550.977,E2 -550.977} C_VEL
LIN {X 0,Y 601.456,Z 159.609,A -85,B 0,C 180,E1 -553.804,E2 -553.804} C_VEL
LIN {X 0,Y 601.428,Z 166.131,A -85,B 0,C 180,E1 -554.876,E2 -554.876} C_VEL
LIN {X 0,Y 601.67,Z 173.375,A -85,B 0,C 180,E1 -554.978,E2 -554.978} C_VEL
LIN {X 0,Y 601.625,Z 273.514,A -85,B 0,C 180,E1 -556.195,E2 -556.195} C_VEL
LIN {X 0,Y 601.576,Z 287.353,A -85,B 0,C 180,E1 -556.515,E2 -556.515} C_VEL
LIN {X 0,Y 601.546,Z 299.362,A -85,B 0,C 180,E1 -556.927,E2 -556.927} C_VEL
LIN {X 0,Y 601.506,Z 311.904,A -85,B 0,C 180,E1 -557.51,E2 -557.51} C_VEL
LIN {X 0,Y 601.462,Z 323.605,A -85,B 0,C 180,E1 -558.214,E2 -558.214} C_VEL
LIN {X 0,Y 601.448,Z 334.089,A -85,B 0,C 180,E1 -559.007,E2 -559.007} C_VEL
LIN {X 0,Y 601.432,Z 342.727,A -85,B 0,C 180,E1 -559.809,E2 -559.809} C_VEL
LIN {X 0,Y 601.385,Z 351.356,A -85,B 0,C 180,E1 -560.786,E2 -560.786} C_VEL
LIN {X 0,Y 601.383,Z 358.465,A -85,B 0,C 180,E1 -561.78,E2 -561.78} C_VEL
LIN {X 0,Y 601.364,Z 363.702,A -85,B 0,C 180,E1 -562.685,E2 -562.685} C_VEL
LIN {X 0,Y 601.344,Z 368.755,A -85,B 0,C 180,E1 -563.779,E2 -563.779} C_VEL
LIN {X 0,Y 601.347,Z 372.523,A -85,B 0,C 180,E1 -564.881,E2 -564.881} C_VEL
LIN {X 0,Y 601.336,Z 374.861,A -85,B 0,C 180,E1 -565.851,E2 -565.851} C_VEL
LIN {X 0,Y 601.332,Z 376.607,A -85,B 0,C 180,E1 -567.117,E2 -567.117} C_VEL
LIN {X 0,Y 601.339,Z 376.966,A -85,B 0,C 180,E1 -567.872,E2 -567.872} C_VEL
LIN {X 0,Y 601.339,Z 376.747,A -85,B 0,C 180,E1 -568.771,E2 -568.771} C_VEL
LIN {X 0,Y 601.346,Z 375.062,A -85,B 0,C 180,E1 -570.134,E2 -570.134} C_VEL
LIN {X 0,Y 601.337,Z 371.815,A -85,B 0,C 180,E1 -571.441,E2 -571.441} C_VEL
LIN {X 0,Y 601.365,Z 367.079,A -85,B 0,C 180,E1 -572.706,E2 -572.706} C_VEL
LIN {X 0,Y 601.381,Z 362.541,A -85,B 0,C 180,E1 -573.62,E2 -573.62} C_VEL
LIN {X 0,Y 601.381,Z 355.65,A -85,B 0,C 180,E1 -574.731,E2 -574.731} C_VEL
LIN {X 0,Y 601.408,Z 347.606,A -85,B 0,C 180,E1 -575.754,E2 -575.754} C_VEL
LIN {X 0,Y 601.412,Z 338.572,A -85,B 0,C 180,E1 -576.687,E2 -576.687} C_VEL
LIN {X 0,Y 601.441,Z 328.537,A -85,B 0,C 180,E1 -577.525,E2 -577.525} C_VEL
LIN {X 0,Y 601.452,Z 317.49,A -85,B 0,C 180,E1 -578.266,E2 -578.266} C_VEL
LIN {X 0,Y 601.519,Z 306.509,A -85,B 0,C 180,E1 -578.852,E2 -578.852} C_VEL
LIN {X 0,Y 601.577,Z 294.084,A -85,B 0,C 180,E1 -579.362,E2 -579.362} C_VEL
LIN {X 0,Y 601.587,Z 281.075,A -85,B 0,C 180,E1 -579.739,E2 -579.739} C_VEL
LIN {X 0,Y 601.611,Z 267.899,A -85,B 0,C 180,E1 -579.98,E2 -579.98} C_VEL
LIN {X 0,Y 601.553,Z 167.04,A -85,B 0,C 180,E1 -581.191,E2 -581.191} C_VEL
LIN {X 0,Y 601.409,Z 166.171,A -85,B 0,C 180,E1 -581.208,E2 -581.208} C_VEL
LIN {X 0,Y 601.444,Z 150.346,A -85,B 0,C 180,E1 -583.817,E2 -583.817} C_VEL
LIN {X 0,Y 601.506,Z 134.746,A -85,B 0,C 180,E1 -586.42,E2 -586.42} C_VEL
LIN {X 0,Y 601.397,Z 128.569,A -85,B 0,C 180,E1 -587.503,E2 -587.503} C_VEL
LIN {X 0,Y 601.381,Z 128.57,A -85,B 0,C 180,E1 -590.002,E2 -590.002} C_VEL
LIN {X 0,Y 601.438,Z 128.572,A -85,B 0,C 180,E1 -592.618,E2 -592.618} C_VEL
LIN {X 0,Y 601.408,Z 128.566,A -85,B 0,C 180,E1 -595.88,E2 -595.88} C_VEL
LIN {X 0,Y 601.418,Z 128.573,A -85,B 0,C 180,E1 -598.547,E2 -598.547} C_VEL
LIN {X 0,Y 601.39,Z 128.567,A -85,B 0,C 180,E1 -601.37,E2 -601.37} C_VEL
LIN {X 0,Y 601.407,Z 128.572,A -85,B 0,C 180,E1 -604.135,E2 -604.135} C_VEL
LIN {X 0,Y 601.381,Z 128.574,A -85,B 0,C 180,E1 -606.588,E2 -606.588} C_VEL
LIN {X 0,Y 601.395,Z 128.567,A -85,B 0,C 180,E1 -609.476,E2 -609.476} C_VEL
LIN {X 0,Y 601.379,Z 128.577,A -85,B 0,C 180,E1 -612.311,E2 -612.311} C_VEL
LIN {X 0,Y 601.378,Z 128.569,A -85,B 0,C 180,E1 -615.101,E2 -615.101} C_VEL
LIN {X 0,Y 601.401,Z 128.573,A -85,B 0,C 180,E1 -617.857,E2 -617.857} C_VEL
LIN {X 0,Y 601.387,Z 128.57,A -85,B 0,C 180,E1 -620.583,E2 -620.583} C_VEL
LIN {X 0,Y 601.377,Z 128.57,A -85,B 0,C 180,E1 -622.614,E2 -622.614} C_VEL
LIN {X 0,Y 601.38,Z 128.57,A -85,B 0,C 180,E1 -625.307,E2 -625.307} C_VEL
LIN {X 0,Y 601.435,Z 128.57,A -85,B 0,C 180,E1 -627.99,E2 -627.99} C_VEL
LIN {X 0,Y 601.366,Z 128.57,A -85,B 0,C 180,E1 -630.669,E2 -630.669} C_VEL
LIN {X 0,Y 601.397,Z 128.566,A -85,B 0,C 180,E1 -632.679,E2 -632.679} C_VEL
LIN {X 0,Y 601.4,Z 128.571,A -85,B 0,C 180,E1 -635.364,E2 -635.364} C_VEL
LIN {X 0,Y 601.429,Z 128.566,A -85,B 0,C 180,E1 -638.06,E2 -638.06} C_VEL
LIN {X 0,Y 601.381,Z 128.57,A -85,B 0,C 180,E1 -640.987,E2 -640.987} C_VEL
LIN {X 0,Y 601.392,Z 128.578,A -85,B 0,C 180,E1 -643.516,E2 -643.516} C_VEL
LIN {X 0,Y 601.388,Z 128.568,A -85,B 0,C 180,E1 -646.288,E2 -646.288} C_VEL
LIN {X 0,Y 601.403,Z 128.571,A -85,B 0,C 180,E1 -649.099,E2 -649.099} C_VEL
LIN {X 0,Y 601.377,Z 128.57,A -85,B 0,C 180,E1 -651.96,E2 -651.96} C_VEL
LIN {X 0,Y 601.378,Z 128.573,A -85,B 0,C 180,E1 -654.879,E2 -654.879} C_VEL
LIN {X 0,Y 601.405,Z 128.574,A -85,B 0,C 180,E1 -657.359,E2 -657.359} C_VEL
LIN {X 0,Y 601.371,Z 128.57,A -85,B 0,C 180,E1 -660.166,E2 -660.166} C_VEL
LIN {X 0,Y 601.389,Z 128.571,A -85,B 0,C 180,E1 -662.71,E2 -662.71} C_VEL
LIN {X 0,Y 601.371,Z 128.58,A -85,B 0,C 180,E1 -665.108,E2 -665.108} C_VEL
LIN {X 0,Y 601.428,Z 128.567,A -85,B 0,C 180,E1 -667.419,E2 -667.419} C_VEL
LIN {X 0,Y 601.372,Z 128.569,A -85,B 0,C 180,E1 -669.997,E2 -669.997} C_VEL
LIN {X 0,Y 601.372,Z 128.576,A -85,B 0,C 180,E1 -672.673,E2 -672.673} C_VEL
LIN {X 0,Y 601.396,Z 128.568,A -85,B 0,C 180,E1 -675.479,E2 -675.479} C_VEL
LIN {X 0,Y 601.403,Z 128.57,A -85,B 0,C 180,E1 -678.408,E2 -678.408} C_VEL
LIN {X 0,Y 601.393,Z 128.575,A -85,B 0,C 180,E1 -680.872,E2 -680.872} C_VEL
LIN {X 0,Y 601.383,Z 128.569,A -85,B 0,C 180,E1 -683.415,E2 -683.415} C_VEL
LIN {X 0,Y 601.392,Z 128.569,A -85,B 0,C 180,E1 -686.069,E2 -686.069} C_VEL
LIN {X 0,Y 601.384,Z 128.571,A -85,B 0,C 180,E1 -689.056,E2 -689.056} C_VEL
LIN {X 0,Y 601.38,Z 128.569,A -85,B 0,C 180,E1 -691.37,E2 -691.37} C_VEL
LIN {X 0,Y 601.392,Z 128.572,A -85,B 0,C 180,E1 -694.135,E2 -694.135} C_VEL
LIN {X 0,Y 601.369,Z 128.578,A -85,B 0,C 180,E1 -696.587,E2 -696.587} C_VEL
LIN {X 0,Y 601.382,Z 128.568,A -85,B 0,C 180,E1 -699.476,E2 -699.476} C_VEL
LIN {X 0,Y 601.357,Z 128.572,A -85,B 0,C 180,E1 -701.606,E2 -701.606} C_VEL
LIN {X 0,Y 601.382,Z 128.576,A -85,B 0,C 180,E1 -704.408,E2 -704.408} C_VEL
LIN {X 0,Y 601.386,Z 128.574,A -85,B 0,C 180,E1 -706.483,E2 -706.483} C_VEL
LIN {X 0,Y 601.349,Z 128.572,A -85,B 0,C 180,E1 -709.222,E2 -709.222} C_VEL
LIN {X 0,Y 601.423,Z 128.571,A -85,B 0,C 180,E1 -711.939,E2 -711.939} C_VEL
LIN {X 0,Y 601.386,Z 128.57,A -85,B 0,C 180,E1 -714.635,E2 -714.635} C_VEL
LIN {X 0,Y 601.391,Z 128.568,A -85,B 0,C 180,E1 -717.321,E2 -717.321} C_VEL
LIN {X 0,Y 601.437,Z 128.571,A -85,B 0,C 180,E1 -720,E2 -720} C_VEL
LIN {X 0,Y 601.388,Z 128.568,A -85,B 0,C 180,E1 -722.679,E2 -722.679} C_VEL
LIN {X 0,Y 601.387,Z 128.571,A -85,B 0,C 180,E1 -725.364,E2 -725.364} C_VEL
LIN {X 0,Y 601.42,Z 128.569,A -85,B 0,C 180,E1 -728.061,E2 -728.061} C_VEL
LIN {X 0,Y 601.368,Z 128.571,A -85,B 0,C 180,E1 -730.988,E2 -730.988} C_VEL
LIN {X 0,Y 601.38,Z 128.576,A -85,B 0,C 180,E1 -733.517,E2 -733.517} C_VEL
LIN {X 0,Y 601.379,Z 128.57,A -85,B 0,C 180,E1 -736.289,E2 -736.289} C_VEL
LIN {X 0,Y 601.392,Z 128.57,A -85,B 0,C 180,E1 -739.1,E2 -739.1} C_VEL
LIN {X 0,Y 601.368,Z 128.573,A -85,B 0,C 180,E1 -741.961,E2 -741.961} C_VEL
LIN {X 0,Y 601.367,Z 128.572,A -85,B 0,C 180,E1 -744.88,E2 -744.88} C_VEL
LIN {X 0,Y 601.391,Z 128.578,A -85,B 0,C 180,E1 -747.36,E2 -747.36} C_VEL
LIN {X 0,Y 601.363,Z 128.571,A -85,B 0,C 180,E1 -750.168,E2 -750.168} C_VEL
LIN {X 0,Y 601.378,Z 128.571,A -85,B 0,C 180,E1 -752.71,E2 -752.71} C_VEL
LIN {X 0,Y 601.36,Z 128.58,A -85,B 0,C 180,E1 -755.108,E2 -755.108} C_VEL
LIN {X 0,Y 601.422,Z 128.569,A -85,B 0,C 180,E1 -757.42,E2 -757.42} C_VEL
LIN {X 0,Y 601.368,Z 128.57,A -85,B 0,C 180,E1 -759.999,E2 -759.999} C_VEL
LIN {X 0,Y 601.36,Z 128.575,A -85,B 0,C 180,E1 -762.675,E2 -762.675} C_VEL
LIN {X 0,Y 601.394,Z 128.57,A -85,B 0,C 180,E1 -765.48,E2 -765.48} C_VEL
LIN {X 0,Y 601.379,Z 128.571,A -85,B 0,C 180,E1 -768.412,E2 -768.412} C_VEL
LIN {X 0,Y 601.39,Z 128.578,A -85,B 0,C 180,E1 -770.873,E2 -770.873} C_VEL
LIN {X 0,Y 601.37,Z 128.572,A -85,B 0,C 180,E1 -773.416,E2 -773.416} C_VEL
LIN {X 0,Y 601.393,Z 128.568,A -85,B 0,C 180,E1 -776.07,E2 -776.07} C_VEL
LIN {X 0,Y 601.383,Z 128.573,A -85,B 0,C 180,E1 -779.057,E2 -779.057} C_VEL
LIN {X 0,Y 601.377,Z 128.57,A -85,B 0,C 180,E1 -781.371,E2 -781.371} C_VEL
LIN {X 0,Y 601.363,Z 128.571,A -85,B 0,C 180,E1 -783.635,E2 -783.635} C_VEL
LIN {X 0,Y 601.386,Z 128.569,A -85,B 0,C 180,E1 -785.857,E2 -785.857} C_VEL
LIN {X 0,Y 601.383,Z 128.678,A -85,B 0,C 180,E1 -787.565,E2 -787.565} C_VEL
LIN {X 0,Y 601.617,Z 137.026,A -85,B 0,C 180,E1 -788.769,E2 -788.769} C_VEL
LIN {X 0,Y 601.554,Z 153.827,A -85,B 0,C 180,E1 -791.144,E2 -791.144} C_VEL
LIN {X 0,Y 601.514,Z 173.546,A -85,B 0,C 180,E1 -793.89,E2 -793.89} C_VEL
LIN {X 0,Y 601.445,Z 194.797,A -85,B 0,C 180,E1 -796.808,E2 -796.808} C_VEL
LIN {X 0,Y 601.651,Z 200.562,A -85,B 0,C 180,E1 -796.898,E2 -796.898} C_VEL
LIN {X 0,Y 601.614,Z 302.981,A -85,B 0,C 180,E1 -798.14,E2 -798.14} C_VEL
LIN {X 0,Y 601.559,Z 316.24,A -85,B 0,C 180,E1 -798.438,E2 -798.438} C_VEL
LIN {X 0,Y 601.538,Z 327.953,A -85,B 0,C 180,E1 -798.827,E2 -798.827} C_VEL
LIN {X 0,Y 601.514,Z 338.937,A -85,B 0,C 180,E1 -799.311,E2 -799.311} C_VEL
LIN {X 0,Y 601.474,Z 349.591,A -85,B 0,C 180,E1 -799.906,E2 -799.906} C_VEL
LIN {X 0,Y 601.448,Z 360.484,A -85,B 0,C 180,E1 -800.67,E2 -800.67} C_VEL
LIN {X 0,Y 601.429,Z 371.118,A -85,B 0,C 180,E1 -801.601,E2 -801.601} C_VEL
LIN {X 0,Y 601.417,Z 378.966,A -85,B 0,C 180,E1 -802.446,E2 -802.446} C_VEL
LIN {X 0,Y 601.369,Z 386.228,A -85,B 0,C 180,E1 -803.398,E2 -803.398} C_VEL
LIN {X 0,Y 601.372,Z 391.869,A -85,B 0,C 180,E1 -804.3,E2 -804.3} C_VEL
LIN {X 0,Y 601.336,Z 396.952,A -85,B 0,C 180,E1 -805.308,E2 -805.308} C_VEL
LIN {X 0,Y 601.368,Z 400.898,A -85,B 0,C 180,E1 -806.315,E2 -806.315} C_VEL
LIN {X 0,Y 601.325,Z 403.81,A -85,B 0,C 180,E1 -807.321,E2 -807.321} C_VEL
LIN {X 0,Y 601.343,Z 405.203,A -85,B 0,C 180,E1 -807.991,E2 -807.991} C_VEL
LIN {X 0,Y 601.339,Z 406.784,A -85,B 0,C 180,E1 -809.331,E2 -809.331} C_VEL
LIN {X 0,Y 601.335,Z 407,A -85,B 0,C 180,E1 -810.001,E2 -810.001} C_VEL
LIN {X 0,Y 601.347,Z 406.184,A -85,B 0,C 180,E1 -811.34,E2 -811.34} C_VEL
LIN {X 0,Y 601.343,Z 405.201,A -85,B 0,C 180,E1 -812.01,E2 -812.01} C_VEL
LIN {X 0,Y 601.325,Z 403.808,A -85,B 0,C 180,E1 -812.68,E2 -812.68} C_VEL
LIN {X 0,Y 601.368,Z 400.894,A -85,B 0,C 180,E1 -813.686,E2 -813.686} C_VEL
LIN {X 0,Y 601.336,Z 396.947,A -85,B 0,C 180,E1 -814.693,E2 -814.693} C_VEL
LIN {X 0,Y 601.373,Z 390.874,A -85,B 0,C 180,E1 -815.87,E2 -815.87} C_VEL
LIN {X 0,Y 601.382,Z 384.232,A -85,B 0,C 180,E1 -816.88,E2 -816.88} C_VEL
LIN {X 0,Y 601.401,Z 375.985,A -85,B 0,C 180,E1 -817.893,E2 -817.893} C_VEL
LIN {X 0,Y 601.436,Z 367.531,A -85,B 0,C 180,E1 -818.738,E2 -818.738} C_VEL
LIN {X 0,Y 601.449,Z 357.086,A -85,B 0,C 180,E1 -819.586,E2 -819.586} C_VEL
LIN {X 0,Y 601.467,Z 346.749,A -85,B 0,C 180,E1 -820.265,E2 -820.265} C_VEL
LIN {X 0,Y 601.538,Z 334.592,A -85,B 0,C 180,E1 -820.896,E2 -820.896} C_VEL
LIN {X 0,Y 601.555,Z 322.202,A -85,B 0,C 180,E1 -821.379,E2 -821.379} C_VEL
LIN {X 0,Y 601.583,Z 309.414,A -85,B 0,C 180,E1 -821.733,E2 -821.733} C_VEL
LIN {X 0,Y 601.621,Z 297.043,A -85,B 0,C 180,E1 -821.946,E2 -821.946} C_VEL
LIN {X 0,Y 601.548,Z 195.88,A -85,B 0,C 180,E1 -823.16,E2 -823.16} C_VEL
LIN {X 0,Y 601.445,Z 194.788,A -85,B 0,C 180,E1 -823.193,E2 -823.193} C_VEL
LIN {X 0,Y 601.515,Z 173.537,A -85,B 0,C 180,E1 -826.111,E2 -826.111} C_VEL
LIN {X 0,Y 601.598,Z 152.129,A -85,B 0,C 180,E1 -829.094,E2 -829.094} C_VEL
LIN {X 0,Y 601.625,Z 131.98,A -85,B 0,C 180,E1 -831.952,E2 -831.952} C_VEL
LIN {X 0,Y 601.374,Z 128.573,A -85,B 0,C 180,E1 -832.462,E2 -832.462} C_VEL
LIN {X 0,Y 601.371,Z 128.573,A -85,B 0,C 180,E1 -834.88,E2 -834.88} C_VEL
LIN {X 0,Y 601.4,Z 128.577,A -85,B 0,C 180,E1 -837.359,E2 -837.359} C_VEL
LIN {X 0,Y 601.372,Z 128.57,A -85,B 0,C 180,E1 -840.168,E2 -840.168} C_VEL
LIN {X 0,Y 601.386,Z 128.571,A -85,B 0,C 180,E1 -842.71,E2 -842.71} C_VEL
LIN {X 0,Y 601.37,Z 128.581,A -85,B 0,C 180,E1 -845.108,E2 -845.108} C_VEL
LIN {X 0,Y 601.431,Z 128.567,A -85,B 0,C 180,E1 -847.42,E2 -847.42} C_VEL
LIN {X 0,Y 601.376,Z 128.569,A -85,B 0,C 180,E1 -849.998,E2 -849.998} C_VEL
LIN {X 0,Y 601.374,Z 128.576,A -85,B 0,C 180,E1 -852.674,E2 -852.674} C_VEL
LIN {X 0,Y 601.402,Z 128.567,A -85,B 0,C 180,E1 -855.48,E2 -855.48} C_VEL
LIN {X 0,Y 601.408,Z 128.57,A -85,B 0,C 180,E1 -858.409,E2 -858.409} C_VEL
LIN {X 0,Y 601.397,Z 128.574,A -85,B 0,C 180,E1 -860.872,E2 -860.872} C_VEL
LIN {X 0,Y 601.387,Z 128.568,A -85,B 0,C 180,E1 -863.416,E2 -863.416} C_VEL
LIN {X 0,Y 601.413,Z 128.568,A -85,B 0,C 180,E1 -866.068,E2 -866.068} C_VEL
LIN {X 0,Y 601.392,Z 128.569,A -85,B 0,C 180,E1 -869.056,E2 -869.056} C_VEL
LIN {X 0,Y 601.389,Z 128.567,A -85,B 0,C 180,E1 -871.371,E2 -871.371} C_VEL
LIN {X 0,Y 601.407,Z 128.572,A -85,B 0,C 180,E1 -874.135,E2 -874.135} C_VEL
LIN {X 0,Y 601.382,Z 128.573,A -85,B 0,C 180,E1 -876.588,E2 -876.588} C_VEL
LIN {X 0,Y 601.398,Z 128.567,A -85,B 0,C 180,E1 -879.477,E2 -879.477} C_VEL
LIN {X 0,Y 601.383,Z 128.575,A -85,B 0,C 180,E1 -882.311,E2 -882.311} C_VEL
LIN {X 0,Y 601.396,Z 128.571,A -85,B 0,C 180,E1 -884.408,E2 -884.408} C_VEL
LIN {X 0,Y 601.402,Z 128.569,A -85,B 0,C 180,E1 -886.484,E2 -886.484} C_VEL
LIN {X 0,Y 601.372,Z 128.571,A -85,B 0,C 180,E1 -889.223,E2 -889.223} C_VEL
LIN {X 0,Y 601.437,Z 128.571,A -85,B 0,C 180,E1 -891.939,E2 -891.939} C_VEL
LIN {X 0,Y 601.399,Z 128.567,A -85,B 0,C 180,E1 -894.636,E2 -894.636} C_VEL
LIN {X 0,Y 601.418,Z 128.568,A -85,B 0,C 180,E1 -897.321,E2 -897.321} C_VEL
LIN {X 0,Y 601.446,Z 128.565,A -85,B 0,C 180,E1 -900,E2 -900} C_VEL
LIN {X 0,Y 601.409,Z 128.566,A -85,B 0,C 180,E1 -902.679,E2 -902.679} C_VEL
LIN {X 0,Y 601.419,Z 128.572,A -85,B 0,C 180,E1 -905.364,E2 -905.364} C_VEL
LIN {X 0,Y 601.432,Z 128.566,A -85,B 0,C 180,E1 -908.061,E2 -908.061} C_VEL
LIN {X 0,Y 601.413,Z 128.74,A -85,B 0,C 180,E1 -908.653,E2 -908.653} C_VEL
LIN {X 0,Y 601.495,Z 141.339,A -85,B 0,C 180,E1 -910.775,E2 -910.775} C_VEL
LIN {X 0,Y 601.481,Z 142.55,A -85,B 0,C 180,E1 -910.977,E2 -910.977} C_VEL
LIN {X 0,Y 600.798,Z 145.55,A -85,B 0,C 180,E1 -911.458,E2 -911.458} C_VEL
LIN {X 0,Y 595.063,Z 155.718,A -85,B 0,C 180,E1 -912.999,E2 -912.999} C_VEL
LIN {X 0,Y 594.424,Z 158.736,A -85,B 0,C 180,E1 -913.487,E2 -913.487} C_VEL
LIN {X 0,Y 594.393,Z 166.279,A -85,B 0,C 180,E1 -914.729,E2 -914.729} C_VEL
LIN {X 0,Y 594.781,Z 171.262,A -85,B 0,C 180,E1 -914.798,E2 -914.798} C_VEL
LIN {X 0,Y 594.695,Z 273.712,A -85,B 0,C 180,E1 -916.058,E2 -916.058} C_VEL
LIN {X 0,Y 594.607,Z 287.82,A -85,B 0,C 180,E1 -916.391,E2 -916.391} C_VEL
LIN {X 0,Y 594.579,Z 300.312,A -85,B 0,C 180,E1 -916.833,E2 -916.833} C_VEL
LIN {X 0,Y 594.515,Z 311.59,A -85,B 0,C 180,E1 -917.367,E2 -917.367} C_VEL
LIN {X 0,Y 594.423,Z 323.369,A -85,B 0,C 180,E1 -918.081,E2 -918.081} C_VEL
LIN {X 0,Y 594.398,Z 333.457,A -85,B 0,C 180,E1 -918.844,E2 -918.844} C_VEL
LIN {X 0,Y 594.36,Z 342.568,A -85,B 0,C 180,E1 -919.694,E2 -919.694} C_VEL
LIN {X 0,Y 594.33,Z 350.551,A -85,B 0,C 180,E1 -920.598,E2 -920.598} C_VEL
LIN {X 0,Y 594.299,Z 358.351,A -85,B 0,C 180,E1 -921.688,E2 -921.688} C_VEL
LIN {X 0,Y 594.278,Z 364.184,A -85,B 0,C 180,E1 -922.714,E2 -922.714} C_VEL
LIN {X 0,Y 594.25,Z 368.681,A -85,B 0,C 180,E1 -923.71,E2 -923.71} C_VEL
LIN {X 0,Y 594.253,Z 372.467,A -85,B 0,C 180,E1 -924.825,E2 -924.825} C_VEL
LIN {X 0,Y 594.228,Z 375.167,A -85,B 0,C 180,E1 -925.991,E2 -925.991} C_VEL
LIN {X 0,Y 594.226,Z 376.195,A -85,B 0,C 180,E1 -926.708,E2 -926.708} C_VEL
LIN {X 0,Y 594.255,Z 376.858,A -85,B 0,C 180,E1 -927.502,E2 -927.502} C_VEL
LIN {X 0,Y 594.224,Z 376.963,A -85,B 0,C 180,E1 -928.235,E2 -928.235} C_VEL
LIN {X 0,Y 594.255,Z 376.595,A -85,B 0,C 180,E1 -929.006,E2 -929.006} C_VEL
LIN {X 0,Y 594.244,Z 374.779,A -85,B 0,C 180,E1 -930.304,E2 -930.304} C_VEL
LIN {X 0,Y 594.242,Z 371.384,A -85,B 0,C 180,E1 -931.621,E2 -931.621} C_VEL
LIN {X 0,Y 594.27,Z 366.495,A -85,B 0,C 180,E1 -932.895,E2 -932.895} C_VEL
LIN {X 0,Y 594.295,Z 360.043,A -85,B 0,C 180,E1 -934.126,E2 -934.126} C_VEL
LIN {X 0,Y 594.316,Z 353.269,A -85,B 0,C 180,E1 -935.138,E2 -935.138} C_VEL
LIN {X 0,Y 594.343,Z 345.954,A -85,B 0,C 180,E1 -936.036,E2 -936.036} C_VEL
LIN {X 0,Y 594.403,Z 337.158,A -85,B 0,C 180,E1 -936.918,E2 -936.918} C_VEL
LIN {X 0,Y 594.429,Z 327.096,A -85,B 0,C 180,E1 -937.744,E2 -937.744} C_VEL
LIN {X 0,Y 594.457,Z 316.056,A -85,B 0,C 180,E1 -938.475,E2 -938.475} C_VEL
LIN {X 0,Y 594.523,Z 304.667,A -85,B 0,C 180,E1 -939.067,E2 -939.067} C_VEL
LIN {X 0,Y 594.62,Z 292.439,A -85,B 0,C 180,E1 -939.552,E2 -939.552} C_VEL
LIN {X 0,Y 594.641,Z 279.782,A -85,B 0,C 180,E1 -939.907,E2 -939.907} C_VEL
LIN {X 0,Y 594.688,Z 266.931,A -85,B 0,C 180,E1 -940.134,E2 -940.134} C_VEL
LIN {X 0,Y 594.594,Z 167.636,A -85,B 0,C 180,E1 -941.34,E2 -941.34} C_VEL
LIN {X 0,Y 594.381,Z 166.099,A -85,B 0,C 180,E1 -941.379,E2 -941.379} C_VEL
LIN {X 0,Y 594.447,Z 149.017,A -85,B 0,C 180,E1 -944.231,E2 -944.231} C_VEL
LIN {X 0,Y 594.532,Z 131.889,A -85,B 0,C 180,E1 -947.131,E2 -947.131} C_VEL
LIN {X 0,Y 594.342,Z 129.449,A -85,B 0,C 180,E1 -947.558,E2 -947.558} C_VEL
LIN {X 0,Y 594.359,Z 129.449,A -85,B 0,C 180,E1 -950.318,E2 -950.318} C_VEL
LIN {X 0,Y 594.381,Z 129.446,A -85,B 0,C 180,E1 -952.912,E2 -952.912} C_VEL
LIN {X 0,Y 594.361,Z 129.444,A -85,B 0,C 180,E1 -955.865,E2 -955.865} C_VEL
LIN {X 0,Y 594.365,Z 129.449,A -85,B 0,C 180,E1 -958.649,E2 -958.649} C_VEL
LIN {X 0,Y 594.345,Z 129.446,A -85,B 0,C 180,E1 -961.05,E2 -961.05} C_VEL
LIN {X 0,Y 594.365,Z 129.448,A -85,B 0,C 180,E1 -964.055,E2 -964.055} C_VEL
LIN {X 0,Y 594.351,Z 129.455,A -85,B 0,C 180,E1 -966.294,E2 -966.294} C_VEL
LIN {X 0,Y 594.375,Z 129.441,A -85,B 0,C 180,E1 -969.223,E2 -969.223} C_VEL
LIN {X 0,Y 594.329,Z 129.456,A -85,B 0,C 180,E1 -972.094,E2 -972.094} C_VEL
LIN {X 0,Y 594.341,Z 129.454,A -85,B 0,C 180,E1 -974.218,E2 -974.218} C_VEL
LIN {X 0,Y 594.369,Z 129.448,A -85,B 0,C 180,E1 -976.32,E2 -976.32} C_VEL
LIN {X 0,Y 594.328,Z 129.447,A -85,B 0,C 180,E1 -979.093,E2 -979.093} C_VEL
LIN {X 0,Y 594.377,Z 129.449,A -85,B 0,C 180,E1 -981.842,E2 -981.842} C_VEL
LIN {X 0,Y 594.362,Z 129.444,A -85,B 0,C 180,E1 -984.571,E2 -984.571} C_VEL
LIN {X 0,Y 594.373,Z 129.443,A -85,B 0,C 180,E1 -987.289,E2 -987.289} C_VEL
LIN {X 0,Y 594.414,Z 129.443,A -85,B 0,C 180,E1 -989.999,E2 -989.999} C_VEL
LIN {X 0,Y 594.366,Z 129.442,A -85,B 0,C 180,E1 -992.71,E2 -992.71} C_VEL
LIN {X 0,Y 594.368,Z 129.448,A -85,B 0,C 180,E1 -995.427,E2 -995.427} C_VEL
LIN {X 0,Y 594.372,Z 129.444,A -85,B 0,C 180,E1 -998.157,E2 -998.157} C_VEL
LIN {X 0,Y 594.35,Z 129.447,A -85,B 0,C 180,E1 -1001.051,E2 -1001.051} C_VEL
LIN {X 0,Y 594.354,Z 129.451,A -85,B 0,C 180,E1 -1003.679,E2 -1003.679} C_VEL
LIN {X 0,Y 594.345,Z 129.445,A -85,B 0,C 180,E1 -1006.486,E2 -1006.486} C_VEL
LIN {X 0,Y 594.354,Z 129.453,A -85,B 0,C 180,E1 -1009.334,E2 -1009.334} C_VEL
LIN {X 0,Y 594.347,Z 129.453,A -85,B 0,C 180,E1 -1011.503,E2 -1011.503} C_VEL
LIN {X 0,Y 594.341,Z 129.446,A -85,B 0,C 180,E1 -1014.447,E2 -1014.447} C_VEL
LIN {X 0,Y 594.359,Z 129.45,A -85,B 0,C 180,E1 -1017.461,E2 -1017.461} C_VEL
LIN {X 0,Y 594.345,Z 129.445,A -85,B 0,C 180,E1 -1020.32,E2 -1020.32} C_VEL
LIN {X 0,Y 594.369,Z 129.449,A -85,B 0,C 180,E1 -1022.95,E2 -1022.95} C_VEL
LIN {X 0,Y 594.309,Z 129.454,A -85,B 0,C 180,E1 -1025.411,E2 -1025.411} C_VEL
LIN {X 0,Y 594.359,Z 129.443,A -85,B 0,C 180,E1 -1027.942,E2 -1027.942} C_VEL
LIN {X 0,Y 594.357,Z 129.451,A -85,B 0,C 180,E1 -1030.819,E2 -1030.819} C_VEL
LIN {X 0,Y 594.338,Z 129.446,A -85,B 0,C 180,E1 -1033.836,E2 -1033.836} C_VEL
LIN {X 0,Y 594.339,Z 129.454,A -85,B 0,C 180,E1 -1036.697,E2 -1036.697} C_VEL
LIN {X 0,Y 594.335,Z 129.447,A -85,B 0,C 180,E1 -1039.43,E2 -1039.43} C_VEL
LIN {X 0,Y 594.372,Z 129.446,A -85,B 0,C 180,E1 -1042.393,E2 -1042.393} C_VEL
LIN {X 0,Y 594.349,Z 129.445,A -85,B 0,C 180,E1 -1045.418,E2 -1045.418} C_VEL
LIN {X 0,Y 594.331,Z 129.447,A -85,B 0,C 180,E1 -1047.85,E2 -1047.85} C_VEL
LIN {X 0,Y 594.331,Z 129.451,A -85,B 0,C 180,E1 -1050.221,E2 -1050.221} C_VEL
LIN {X 0,Y 594.348,Z 129.445,A -85,B 0,C 180,E1 -1053.298,E2 -1053.298} C_VEL
LIN {X 0,Y 594.327,Z 129.447,A -85,B 0,C 180,E1 -1055.577,E2 -1055.577} C_VEL
LIN {X 0,Y 594.341,Z 129.454,A -85,B 0,C 180,E1 -1058.495,E2 -1058.495} C_VEL
LIN {X 0,Y 594.335,Z 129.446,A -85,B 0,C 180,E1 -1061.381,E2 -1061.381} C_VEL
LIN {X 0,Y 594.33,Z 129.456,A -85,B 0,C 180,E1 -1064.218,E2 -1064.218} C_VEL
LIN {X 0,Y 594.352,Z 129.453,A -85,B 0,C 180,E1 -1066.32,E2 -1066.32} C_VEL
LIN {X 0,Y 594.316,Z 129.449,A -85,B 0,C 180,E1 -1069.093,E2 -1069.093} C_VEL
LIN {X 0,Y 594.364,Z 129.448,A -85,B 0,C 180,E1 -1071.842,E2 -1071.842} C_VEL
LIN {X 0,Y 594.357,Z 129.446,A -85,B 0,C 180,E1 -1074.572,E2 -1074.572} C_VEL
LIN {X 0,Y 594.359,Z 129.444,A -85,B 0,C 180,E1 -1077.289,E2 -1077.289} C_VEL
LIN {X 0,Y 594.405,Z 129.447,A -85,B 0,C 180,E1 -1080,E2 -1080} C_VEL
LIN {X 0,Y 594.356,Z 129.444,A -85,B 0,C 180,E1 -1082.711,E2 -1082.711} C_VEL
LIN {X 0,Y 594.356,Z 129.447,A -85,B 0,C 180,E1 -1085.428,E2 -1085.428} C_VEL
LIN {X 0,Y 594.362,Z 129.447,A -85,B 0,C 180,E1 -1088.157,E2 -1088.157} C_VEL
LIN {X 0,Y 594.337,Z 129.447,A -85,B 0,C 180,E1 -1091.052,E2 -1091.052} C_VEL
LIN {X 0,Y 594.347,Z 129.455,A -85,B 0,C 180,E1 -1093.68,E2 -1093.68} C_VEL
LIN {X 0,Y 594.309,Z 129.449,A -85,B 0,C 180,E1 -1096.695,E2 -1096.695} C_VEL
LIN {X 0,Y 594.343,Z 129.452,A -85,B 0,C 180,E1 -1099.335,E2 -1099.335} C_VEL
LIN {X 0,Y 594.337,Z 129.456,A -85,B 0,C 180,E1 -1101.504,E2 -1101.504} C_VEL
LIN {X 0,Y 594.332,Z 129.446,A -85,B 0,C 180,E1 -1104.449,E2 -1104.449} C_VEL
LIN {X 0,Y 594.344,Z 129.446,A -85,B 0,C 180,E1 -1106.701,E2 -1106.701} C_VEL
LIN {X 0,Y 594.325,Z 129.451,A -85,B 0,C 180,E1 -1109.779,E2 -1109.779} C_VEL
LIN {X 0,Y 594.326,Z 129.447,A -85,B 0,C 180,E1 -1112.15,E2 -1112.15} C_VEL
LIN {X 0,Y 594.346,Z 129.446,A -85,B 0,C 180,E1 -1114.582,E2 -1114.582} C_VEL
LIN {X 0,Y 594.367,Z 129.445,A -85,B 0,C 180,E1 -1117.607,E2 -1117.607} C_VEL
LIN {X 0,Y 594.331,Z 129.449,A -85,B 0,C 180,E1 -1120.57,E2 -1120.57} C_VEL
LIN {X 0,Y 594.333,Z 129.452,A -85,B 0,C 180,E1 -1123.303,E2 -1123.303} C_VEL
LIN {X 0,Y 594.335,Z 129.446,A -85,B 0,C 180,E1 -1126.164,E2 -1126.164} C_VEL
LIN {X 0,Y 594.351,Z 129.45,A -85,B 0,C 180,E1 -1129.181,E2 -1129.181} C_VEL
LIN {X 0,Y 594.338,Z 129.446,A -85,B 0,C 180,E1 -1132.057,E2 -1132.057} C_VEL
LIN {X 0,Y 594.302,Z 129.459,A -85,B 0,C 180,E1 -1134.684,E2 -1134.684} C_VEL
LIN {X 0,Y 594.335,Z 129.451,A -85,B 0,C 180,E1 -1137.095,E2 -1137.095} C_VEL
LIN {X 0,Y 594.341,Z 129.445,A -85,B 0,C 180,E1 -1139.68,E2 -1139.68} C_VEL
LIN {X 0,Y 594.336,Z 129.455,A -85,B 0,C 180,E1 -1142.538,E2 -1142.538} C_VEL
LIN {X 0,Y 594.346,Z 129.453,A -85,B 0,C 180,E1 -1144.806,E2 -1144.806} C_VEL
LIN {X 0,Y 594.341,Z 129.621,A -85,B 0,C 180,E1 -1147.422,E2 -1147.422} C_VEL
LIN {X 0,Y 594.731,Z 135.766,A -85,B 0,C 180,E1 -1148.329,E2 -1148.329} C_VEL
LIN {X 0,Y 594.596,Z 155.314,A -85,B 0,C 180,E1 -1151.126,E2 -1151.126} C_VEL
LIN {X 0,Y 594.518,Z 174.805,A -85,B 0,C 180,E1 -1153.872,E2 -1153.872} C_VEL
LIN {X 0,Y 594.46,Z 195.196,A -85,B 0,C 180,E1 -1156.672,E2 -1156.672} C_VEL
LIN {X 0,Y 594.73,Z 205.928,A -85,B 0,C 180,E1 -1156.808,E2 -1156.808} C_VEL
LIN {X 0,Y 594.665,Z 302.98,A -85,B 0,C 180,E1 -1158,E2 -1158} C_VEL
LIN {X 0,Y 594.601,Z 316.241,A -85,B 0,C 180,E1 -1158.301,E2 -1158.301} C_VEL
LIN {X 0,Y 594.571,Z 328.577,A -85,B 0,C 180,E1 -1158.718,E2 -1158.718} C_VEL
LIN {X 0,Y 594.536,Z 340.643,A -85,B 0,C 180,E1 -1159.271,E2 -1159.271} C_VEL
LIN {X 0,Y 594.477,Z 352.21,A -85,B 0,C 180,E1 -1159.958,E2 -1159.958} C_VEL
LIN {X 0,Y 594.414,Z 362.605,A -85,B 0,C 180,E1 -1160.73,E2 -1160.73} C_VEL
LIN {X 0,Y 594.383,Z 371.119,A -85,B 0,C 180,E1 -1161.501,E2 -1161.501} C_VEL
LIN {X 0,Y 594.347,Z 378.966,A -85,B 0,C 180,E1 -1162.356,E2 -1162.356} C_VEL
LIN {X 0,Y 594.282,Z 386.816,A -85,B 0,C 180,E1 -1163.409,E2 -1163.409} C_VEL
LIN {X 0,Y 594.289,Z 393.683,A -85,B 0,C 180,E1 -1164.572,E2 -1164.572} C_VEL
LIN {X 0,Y 594.27,Z 398.374,A -85,B 0,C 180,E1 -1165.592,E2 -1165.592} C_VEL
LIN {X 0,Y 594.267,Z 401.958,A -85,B 0,C 180,E1 -1166.611,E2 -1166.611} C_VEL
LIN {X 0,Y 594.226,Z 403.81,A -85,B 0,C 180,E1 -1167.289,E2 -1167.289} C_VEL
LIN {X 0,Y 594.242,Z 405.202,A -85,B 0,C 180,E1 -1167.967,E2 -1167.967} C_VEL
LIN {X 0,Y 594.239,Z 406.785,A -85,B 0,C 180,E1 -1169.323,E2 -1169.323} C_VEL
LIN {X 0,Y 594.236,Z 407,A -85,B 0,C 180,E1 -1170.001,E2 -1170.001} C_VEL
LIN {X 0,Y 594.247,Z 406.184,A -85,B 0,C 180,E1 -1171.356,E2 -1171.356} C_VEL
LIN {X 0,Y 594.242,Z 405.2,A -85,B 0,C 180,E1 -1172.034,E2 -1172.034} C_VEL
LIN {X 0,Y 594.226,Z 403.808,A -85,B 0,C 180,E1 -1172.712,E2 -1172.712} C_VEL
LIN {X 0,Y 594.289,Z 400.894,A -85,B 0,C 180,E1 -1173.73,E2 -1173.73} C_VEL
LIN {X 0,Y 594.241,Z 396.947,A -85,B 0,C 180,E1 -1174.749,E2 -1174.749} C_VEL
LIN {X 0,Y 594.305,Z 390.874,A -85,B 0,C 180,E1 -1175.94,E2 -1175.94} C_VEL
LIN {X 0,Y 594.308,Z 384.232,A -85,B 0,C 180,E1 -1176.963,E2 -1176.963} C_VEL
LIN {X 0,Y 594.359,Z 375.985,A -85,B 0,C 180,E1 -1177.987,E2 -1177.987} C_VEL
LIN {X 0,Y 594.382,Z 367.531,A -85,B 0,C 180,E1 -1178.843,E2 -1178.843} C_VEL
LIN {X 0,Y 594.432,Z 357.087,A -85,B 0,C 180,E1 -1179.7,E2 -1179.7} C_VEL
LIN {X 0,Y 594.482,Z 346.749,A -85,B 0,C 180,E1 -1180.387,E2 -1180.387} C_VEL
LIN {X 0,Y 594.558,Z 335.722,A -85,B 0,C 180,E1 -1180.973,E2 -1180.973} C_VEL
LIN {X 0,Y 594.58,Z 323.698,A -85,B 0,C 180,E1 -1181.465,E2 -1181.465} C_VEL
LIN {X 0,Y 594.625,Z 310.327,A -85,B 0,C 180,E1 -1181.851,E2 -1181.851} C_VEL
LIN {X 0,Y 594.699,Z 297.043,A -85,B 0,C 180,E1 -1182.087,E2 -1182.087} C_VEL
LIN {X 0,Y 594.685,Z 196.886,A -85,B 0,C 180,E1 -1183.302,E2 -1183.302} C_VEL
LIN {X 0,Y 594.423,Z 194.788,A -85,B 0,C 180,E1 -1183.352,E2 -1183.352} C_VEL
LIN {X 0,Y 594.524,Z 173.537,A -85,B 0,C 180,E1 -1186.306,E2 -1186.306} C_VEL
LIN {X 0,Y 594.632,Z 153.721,A -85,B 0,C 180,E1 -1189.099,E2 -1189.099} C_VEL
LIN {X 0,Y 594.705,Z 133.239,A -85,B 0,C 180,E1 -1192.038,E2 -1192.038} C_VEL
LIN {X 0,Y 594.306,Z 129.455,A -85,B 0,C 180,E1 -1192.613,E2 -1192.613} C_VEL
LIN {X 0,Y 594.327,Z 129.455,A -85,B 0,C 180,E1 -1195.196,E2 -1195.196} C_VEL
LIN {X 0,Y 594.346,Z 129.452,A -85,B 0,C 180,E1 -1197.519,E2 -1197.519} C_VEL
LIN {X 0,Y 594.347,Z 129.445,A -85,B 0,C 180,E1 -1200.321,E2 -1200.321} C_VEL
LIN {X 0,Y 594.341,Z 129.452,A -85,B 0,C 180,E1 -1202.953,E2 -1202.953} C_VEL
LIN {X 0,Y 594.305,Z 129.455,A -85,B 0,C 180,E1 -1205.413,E2 -1205.413} C_VEL
LIN {X 0,Y 594.347,Z 129.445,A -85,B 0,C 180,E1 -1207.944,E2 -1207.944} C_VEL
LIN {X 0,Y 594.36,Z 129.451,A -85,B 0,C 180,E1 -1210.82,E2 -1210.82} C_VEL
LIN {X 0,Y 594.343,Z 129.445,A -85,B 0,C 180,E1 -1213.837,E2 -1213.837} C_VEL
LIN {X 0,Y 594.344,Z 129.453,A -85,B 0,C 180,E1 -1216.698,E2 -1216.698} C_VEL
LIN {X 0,Y 594.342,Z 129.446,A -85,B 0,C 180,E1 -1219.431,E2 -1219.431} C_VEL
LIN {X 0,Y 594.378,Z 129.447,A -85,B 0,C 180,E1 -1222.394,E2 -1222.394} C_VEL
LIN {X 0,Y 594.359,Z 129.444,A -85,B 0,C 180,E1 -1225.419,E2 -1225.419} C_VEL
LIN {X 0,Y 594.34,Z 129.447,A -85,B 0,C 180,E1 -1227.851,E2 -1227.851} C_VEL
LIN {X 0,Y 594.341,Z 129.452,A -85,B 0,C 180,E1 -1230.222,E2 -1230.222} C_VEL
LIN {X 0,Y 594.357,Z 129.444,A -85,B 0,C 180,E1 -1233.299,E2 -1233.299} C_VEL
LIN {X 0,Y 594.342,Z 129.446,A -85,B 0,C 180,E1 -1235.577,E2 -1235.577} C_VEL
LIN {X 0,Y 594.35,Z 129.45,A -85,B 0,C 180,E1 -1238.496,E2 -1238.496} C_VEL
LIN {X 0,Y 594.35,Z 129.445,A -85,B 0,C 180,E1 -1241.381,E2 -1241.381} C_VEL
LIN {X 0,Y 594.346,Z 129.453,A -85,B 0,C 180,E1 -1244.219,E2 -1244.219} C_VEL
LIN {X 0,Y 594.372,Z 129.447,A -85,B 0,C 180,E1 -1246.321,E2 -1246.321} C_VEL
LIN {X 0,Y 594.347,Z 129.445,A -85,B 0,C 180,E1 -1249.094,E2 -1249.094} C_VEL
LIN {X 0,Y 594.38,Z 129.451,A -85,B 0,C 180,E1 -1251.843,E2 -1251.843} C_VEL
LIN {X 0,Y 594.37,Z 129.443,A -85,B 0,C 180,E1 -1254.572,E2 -1254.572} C_VEL
LIN {X 0,Y 594.384,Z 129.444,A -85,B 0,C 180,E1 -1257.289,E2 -1257.289} C_VEL
LIN {X 0,Y 594.415,Z 129.441,A -85,B 0,C 180,E1 -1260,E2 -1260} C_VEL
LIN {X 0,Y 594.379,Z 129.442,A -85,B 0,C 180,E1 -1262.711,E2 -1262.711} C_VEL
LIN {X 0,Y 594.384,Z 129.45,A -85,B 0,C 180,E1 -1265.428,E2 -1265.428} C_VEL
LIN {X 0,Y 594.372,Z 129.446,A -85,B 0,C 180,E1 -1268.5,E2 -1268.5} C_VEL
LIN {X 0,Y 594.535,Z 136.223,A -85,B 0,C 180,E1 -1269.698,E2 -1269.698} C_VEL
LIN {X 0,Y 594.452,Z 153.632,A -85,B 0,C 180,E1 -1272.634,E2 -1272.634} C_VEL
LIN {X 0,Y 594.424,Z 158.736,A -85,B 0,C 180,E1 -1273.487,E2 -1273.487} C_VEL
LIN {X 0,Y 593.811,Z 161.001,A -85,B 0,C 180,E1 -1273.817,E2 -1273.817} C_VEL
LIN {X 0,Y 592.347,Z 163.57,A -85,B 0,C 180,E1 -1274.106,E2 -1274.106} C_VEL
LIN {X 0,Y 589.998,Z 167.492,A -85,B 0,C 180,E1 -1274.416,E2 -1274.416} C_VEL
LIN {X 0,Y 588.333,Z 171.542,A -85,B 0,C 180,E1 -1274.608,E2 -1274.608} C_VEL
LIN {X 0,Y 587.859,Z 174.802,A -85,B 0,C 180,E1 -1274.683,E2 -1274.683} C_VEL
LIN {X 0,Y 587.731,Z 272.637,A -85,B 0,C 180,E1 -1275.897,E2 -1275.897} C_VEL
LIN {X 0,Y 587.644,Z 285.703,A -85,B 0,C 180,E1 -1276.189,E2 -1276.189} C_VEL
LIN {X 0,Y 587.608,Z 297.606,A -85,B 0,C 180,E1 -1276.592,E2 -1276.592} C_VEL
LIN {X 0,Y 587.557,Z 309.786,A -85,B 0,C 180,E1 -1277.142,E2 -1277.142} C_VEL
LIN {X 0,Y 587.45,Z 320.406,A -85,B 0,C 180,E1 -1277.763,E2 -1277.763} C_VEL
LIN {X 0,Y 587.404,Z 330.425,A -85,B 0,C 180,E1 -1278.485,E2 -1278.485} C_VEL
LIN {X 0,Y 587.339,Z 340.88,A -85,B 0,C 180,E1 -1279.42,E2 -1279.42} C_VEL
LIN {X 0,Y 587.252,Z 348.93,A -85,B 0,C 180,E1 -1280.308,E2 -1280.308} C_VEL
LIN {X 0,Y 587.243,Z 357.049,A -85,B 0,C 180,E1 -1281.409,E2 -1281.409} C_VEL
LIN {X 0,Y 587.187,Z 363.506,A -85,B 0,C 180,E1 -1282.52,E2 -1282.52} C_VEL
LIN {X 0,Y 587.174,Z 368.603,A -85,B 0,C 180,E1 -1283.639,E2 -1283.639} C_VEL
LIN {X 0,Y 587.175,Z 372.41,A -85,B 0,C 180,E1 -1284.767,E2 -1284.767} C_VEL
LIN {X 0,Y 587.121,Z 375.442,A -85,B 0,C 180,E1 -1286.133,E2 -1286.133} C_VEL
LIN {X 0,Y 587.133,Z 376.586,A -85,B 0,C 180,E1 -1287.056,E2 -1287.056} C_VEL
LIN {X 0,Y 587.148,Z 376.957,A -85,B 0,C 180,E1 -1287.828,E2 -1287.828} C_VEL
LIN {X 0,Y 587.168,Z 376.524,A -85,B 0,C 180,E1 -1289.101,E2 -1289.101} C_VEL
LIN {X 0,Y 587.158,Z 374.473,A -85,B 0,C 180,E1 -1290.479,E2 -1290.479} C_VEL
LIN {X 0,Y 587.144,Z 370.935,A -85,B 0,C 180,E1 -1291.803,E2 -1291.803} C_VEL
LIN {X 0,Y 587.175,Z 365.887,A -85,B 0,C 180,E1 -1293.086,E2 -1293.086} C_VEL
LIN {X 0,Y 587.2,Z 359.859,A -85,B 0,C 180,E1 -1294.231,E2 -1294.231} C_VEL
LIN {X 0,Y 587.28,Z 352.756,A -85,B 0,C 180,E1 -1295.294,E2 -1295.294} C_VEL
LIN {X 0,Y 587.287,Z 344.189,A -85,B 0,C 180,E1 -1296.325,E2 -1296.325} C_VEL
LIN {X 0,Y 587.361,Z 335.484,A -85,B 0,C 180,E1 -1297.175,E2 -1297.175} C_VEL
LIN {X 0,Y 587.414,Z 325.01,A -85,B 0,C 180,E1 -1298.017,E2 -1298.017} C_VEL
LIN {X 0,Y 587.495,Z 313.553,A -85,B 0,C 180,E1 -1298.742,E2 -1298.742} C_VEL
LIN {X 0,Y 587.594,Z 301.531,A -85,B 0,C 180,E1 -1299.34,E2 -1299.34} C_VEL
LIN {X 0,Y 587.649,Z 288.819,A -85,B 0,C 180,E1 -1299.807,E2 -1299.807} C_VEL
LIN {X 0,Y 587.732,Z 275.602,A -85,B 0,C 180,E1 -1300.14,E2 -1300.14} C_VEL
LIN {X 0,Y 587.77,Z 254.751,A -85,B 0,C 180,E1 -1300.428,E2 -1300.428} C_VEL
LIN {X 0,Y 587.707,Z 168.568,A -85,B 0,C 180,E1 -1301.488,E2 -1301.488} C_VEL
LIN {X 0,Y 587.364,Z 166.126,A -85,B 0,C 180,E1 -1301.537,E2 -1301.537} C_VEL
LIN {X 0,Y 587.441,Z 148.724,A -85,B 0,C 180,E1 -1304.479,E2 -1304.479} C_VEL
LIN {X 0,Y 587.524,Z 132.592,A -85,B 0,C 180,E1 -1307.246,E2 -1307.246} C_VEL
LIN {X 0,Y 587.298,Z 130.327,A -85,B 0,C 180,E1 -1307.691,E2 -1307.691} C_VEL
LIN {X 0,Y 587.32,Z 130.33,A -85,B 0,C 180,E1 -1310.638,E2 -1310.638} C_VEL
LIN {X 0,Y 587.32,Z 130.321,A -85,B 0,C 180,E1 -1313.297,E2 -1313.297} C_VEL
LIN {X 0,Y 587.324,Z 130.32,A -85,B 0,C 180,E1 -1315.777,E2 -1315.777} C_VEL
LIN {X 0,Y 587.338,Z 130.324,A -85,B 0,C 180,E1 -1318.23,E2 -1318.23} C_VEL
LIN {X 0,Y 587.305,Z 130.325,A -85,B 0,C 180,E1 -1320.876,E2 -1320.876} C_VEL
LIN {X 0,Y 587.31,Z 130.324,A -85,B 0,C 180,E1 -1323.83,E2 -1323.83} C_VEL
LIN {X 0,Y 587.294,Z 130.326,A -85,B 0,C 180,E1 -1326.74,E2 -1326.74} C_VEL
LIN {X 0,Y 587.305,Z 130.324,A -85,B 0,C 180,E1 -1329.694,E2 -1329.694} C_VEL
LIN {X 0,Y 587.277,Z 130.329,A -85,B 0,C 180,E1 -1332.591,E2 -1332.591} C_VEL
LIN {X 0,Y 587.319,Z 130.321,A -85,B 0,C 180,E1 -1335.446,E2 -1335.446} C_VEL
LIN {X 0,Y 587.318,Z 130.327,A -85,B 0,C 180,E1 -1338.262,E2 -1338.262} C_VEL
LIN {X 0,Y 587.282,Z 130.325,A -85,B 0,C 180,E1 -1341.05,E2 -1341.05} C_VEL
LIN {X 0,Y 587.312,Z 130.329,A -85,B 0,C 180,E1 -1343.817,E2 -1343.817} C_VEL
LIN {X 0,Y 587.306,Z 130.332,A -85,B 0,C 180,E1 -1345.882,E2 -1345.882} C_VEL
LIN {X 0,Y 587.372,Z 130.322,A -85,B 0,C 180,E1 -1347.942,E2 -1347.942} C_VEL
LIN {X 0,Y 587.383,Z 130.319,A -85,B 0,C 180,E1 -1349.999,E2 -1349.999} C_VEL
LIN {X 0,Y 587.335,Z 130.318,A -85,B 0,C 180,E1 -1352.743,E2 -1352.743} C_VEL
LIN {X 0,Y 587.336,Z 130.325,A -85,B 0,C 180,E1 -1355.493,E2 -1355.493} C_VEL
LIN {X 0,Y 587.328,Z 130.321,A -85,B 0,C 180,E1 -1358.255,E2 -1358.255} C_VEL
LIN {X 0,Y 587.319,Z 130.323,A -85,B 0,C 180,E1 -1361.116,E2 -1361.116} C_VEL
LIN {X 0,Y 587.304,Z 130.323,A -85,B 0,C 180,E1 -1364.234,E2 -1364.234} C_VEL
LIN {X 0,Y 587.295,Z 130.324,A -85,B 0,C 180,E1 -1366.795,E2 -1366.795} C_VEL
LIN {X 0,Y 587.297,Z 130.33,A -85,B 0,C 180,E1 -1369.576,E2 -1369.576} C_VEL
LIN {X 0,Y 587.295,Z 130.327,A -85,B 0,C 180,E1 -1371.775,E2 -1371.775} C_VEL
LIN {X 0,Y 587.297,Z 130.325,A -85,B 0,C 180,E1 -1374.76,E2 -1374.76} C_VEL
LIN {X 0,Y 587.296,Z 130.326,A -85,B 0,C 180,E1 -1377.681,E2 -1377.681} C_VEL
LIN {X 0,Y 587.287,Z 130.325,A -85,B 0,C 180,E1 -1380.501,E2 -1380.501} C_VEL
LIN {X 0,Y 587.317,Z 130.326,A -85,B 0,C 180,E1 -1383.397,E2 -1383.397} C_VEL
LIN {X 0,Y 587.262,Z 130.327,A -85,B 0,C 180,E1 -1385.901,E2 -1385.901} C_VEL
LIN {X 0,Y 587.307,Z 130.324,A -85,B 0,C 180,E1 -1388.48,E2 -1388.48} C_VEL
LIN {X 0,Y 587.305,Z 130.329,A -85,B 0,C 180,E1 -1391.159,E2 -1391.159} C_VEL
LIN {X 0,Y 587.299,Z 130.323,A -85,B 0,C 180,E1 -1394.11,E2 -1394.11} C_VEL
LIN {X 0,Y 587.281,Z 130.332,A -85,B 0,C 180,E1 -1396.99,E2 -1396.99} C_VEL
LIN {X 0,Y 587.287,Z 130.324,A -85,B 0,C 180,E1 -1399.743,E2 -1399.743} C_VEL
LIN {X 0,Y 587.326,Z 130.324,A -85,B 0,C 180,E1 -1402.39,E2 -1402.39} C_VEL
LIN {X 0,Y 587.315,Z 130.321,A -85,B 0,C 180,E1 -1405.656,E2 -1405.656} C_VEL
LIN {X 0,Y 587.326,Z 130.323,A -85,B 0,C 180,E1 -1408.23,E2 -1408.23} C_VEL
LIN {X 0,Y 587.294,Z 130.328,A -85,B 0,C 180,E1 -1410.875,E2 -1410.875} C_VEL
LIN {X 0,Y 587.297,Z 130.324,A -85,B 0,C 180,E1 -1413.83,E2 -1413.83} C_VEL
LIN {X 0,Y 587.281,Z 130.33,A -85,B 0,C 180,E1 -1416.739,E2 -1416.739} C_VEL
LIN {X 0,Y 587.293,Z 130.325,A -85,B 0,C 180,E1 -1419.694,E2 -1419.694} C_VEL
LIN {X 0,Y 587.267,Z 130.33,A -85,B 0,C 180,E1 -1421.871,E2 -1421.871} C_VEL
LIN {X 0,Y 587.29,Z 130.327,A -85,B 0,C 180,E1 -1424.736,E2 -1424.736} C_VEL
LIN {X 0,Y 587.264,Z 130.328,A -85,B 0,C 180,E1 -1426.857,E2 -1426.857} C_VEL
LIN {X 0,Y 587.313,Z 130.324,A -85,B 0,C 180,E1 -1429.659,E2 -1429.659} C_VEL
LIN {X 0,Y 587.303,Z 130.327,A -85,B 0,C 180,E1 -1432.436,E2 -1432.436} C_VEL
LIN {X 0,Y 587.315,Z 130.321,A -85,B 0,C 180,E1 -1435.195,E2 -1435.195} C_VEL
LIN {X 0,Y 587.366,Z 130.324,A -85,B 0,C 180,E1 -1437.943,E2 -1437.943} C_VEL
LIN {X 0,Y 587.373,Z 130.323,A -85,B 0,C 180,E1 -1440,E2 -1440} C_VEL
LIN {X 0,Y 587.325,Z 130.32,A -85,B 0,C 180,E1 -1442.743,E2 -1442.743} C_VEL
LIN {X 0,Y 587.325,Z 130.324,A -85,B 0,C 180,E1 -1445.493,E2 -1445.493} C_VEL
LIN {X 0,Y 587.318,Z 130.323,A -85,B 0,C 180,E1 -1448.256,E2 -1448.256} C_VEL
LIN {X 0,Y 587.307,Z 130.323,A -85,B 0,C 180,E1 -1451.117,E2 -1451.117} C_VEL
LIN {X 0,Y 587.309,Z 130.323,A -85,B 0,C 180,E1 -1454.241,E2 -1454.241} C_VEL
LIN {X 0,Y 587.284,Z 130.325,A -85,B 0,C 180,E1 -1456.796,E2 -1456.796} C_VEL
LIN {X 0,Y 587.287,Z 130.334,A -85,B 0,C 180,E1 -1459.577,E2 -1459.577} C_VEL
LIN {X 0,Y 587.285,Z 130.33,A -85,B 0,C 180,E1 -1461.776,E2 -1461.776} C_VEL
LIN {X 0,Y 587.288,Z 130.325,A -85,B 0,C 180,E1 -1464.761,E2 -1464.761} C_VEL
LIN {X 0,Y 587.287,Z 130.329,A -85,B 0,C 180,E1 -1467.682,E2 -1467.682} C_VEL
LIN {X 0,Y 587.279,Z 130.326,A -85,B 0,C 180,E1 -1470.502,E2 -1470.502} C_VEL
LIN {X 0,Y 587.322,Z 130.328,A -85,B 0,C 180,E1 -1473.111,E2 -1473.111} C_VEL
LIN {X 0,Y 587.254,Z 130.329,A -85,B 0,C 180,E1 -1475.903,E2 -1475.903} C_VEL
LIN {X 0,Y 587.292,Z 130.325,A -85,B 0,C 180,E1 -1478.482,E2 -1478.482} C_VEL
LIN {X 0,Y 587.299,Z 130.332,A -85,B 0,C 180,E1 -1481.16,E2 -1481.16} C_VEL
LIN {X 0,Y 587.296,Z 130.323,A -85,B 0,C 180,E1 -1484.111,E2 -1484.111} C_VEL
LIN {X 0,Y 587.276,Z 130.336,A -85,B 0,C 180,E1 -1486.991,E2 -1486.991} C_VEL
LIN {X 0,Y 587.285,Z 130.325,A -85,B 0,C 180,E1 -1489.744,E2 -1489.744} C_VEL
LIN {X 0,Y 587.323,Z 130.323,A -85,B 0,C 180,E1 -1492.392,E2 -1492.392} C_VEL
LIN {X 0,Y 587.307,Z 130.322,A -85,B 0,C 180,E1 -1495.777,E2 -1495.777} C_VEL
LIN {X 0,Y 587.295,Z 130.326,A -85,B 0,C 180,E1 -1498.229,E2 -1498.229} C_VEL
LIN {X 0,Y 587.294,Z 130.33,A -85,B 0,C 180,E1 -1500.877,E2 -1500.877} C_VEL
LIN {X 0,Y 587.291,Z 130.325,A -85,B 0,C 180,E1 -1503.833,E2 -1503.833} C_VEL
LIN {X 0,Y 587.282,Z 130.334,A -85,B 0,C 180,E1 -1506.74,E2 -1506.74} C_VEL
LIN {X 0,Y 587.283,Z 130.447,A -85,B 0,C 180,E1 -1507.269,E2 -1507.269} C_VEL
LIN {X 0,Y 587.77,Z 135.75,A -85,B 0,C 180,E1 -1508.059,E2 -1508.059} C_VEL
LIN {X 0,Y 587.67,Z 155.134,A -85,B 0,C 180,E1 -1510.869,E2 -1510.869} C_VEL
LIN {X 0,Y 587.527,Z 174.805,A -85,B 0,C 180,E1 -1513.674,E2 -1513.674} C_VEL
LIN {X 0,Y 587.381,Z 194.797,A -85,B 0,C 180,E1 -1516.486,E2 -1516.486} C_VEL
LIN {X 0,Y 587.839,Z 198.773,A -85,B 0,C 180,E1 -1516.563,E2 -1516.563} C_VEL
LIN {X 0,Y 587.728,Z 302.98,A -85,B 0,C 180,E1 -1517.856,E2 -1517.856} C_VEL
LIN {X 0,Y 587.667,Z 316.242,A -85,B 0,C 180,E1 -1518.161,E2 -1518.161} C_VEL
LIN {X 0,Y 587.599,Z 328.783,A -85,B 0,C 180,E1 -1518.591,E2 -1518.591} C_VEL
LIN {X 0,Y 587.536,Z 340.641,A -85,B 0,C 180,E1 -1519.141,E2 -1519.141} C_VEL
LIN {X 0,Y 587.464,Z 352.212,A -85,B 0,C 180,E1 -1519.837,E2 -1519.837} C_VEL
LIN {X 0,Y 587.394,Z 362.607,A -85,B 0,C 180,E1 -1520.618,E2 -1520.618} C_VEL
LIN {X 0,Y 587.321,Z 371.119,A -85,B 0,C 180,E1 -1521.398,E2 -1521.398} C_VEL
LIN {X 0,Y 587.273,Z 378.966,A -85,B 0,C 180,E1 -1522.263,E2 -1522.263} C_VEL
LIN {X 0,Y 587.229,Z 385.473,A -85,B 0,C 180,E1 -1523.127,E2 -1523.127} C_VEL
LIN {X 0,Y 587.237,Z 391.87,A -85,B 0,C 180,E1 -1524.162,E2 -1524.162} C_VEL
LIN {X 0,Y 587.147,Z 396.952,A -85,B 0,C 180,E1 -1525.194,E2 -1525.194} C_VEL
LIN {X 0,Y 587.213,Z 400.897,A -85,B 0,C 180,E1 -1526.226,E2 -1526.226} C_VEL
LIN {X 0,Y 587.132,Z 403.81,A -85,B 0,C 180,E1 -1527.256,E2 -1527.256} C_VEL
LIN {X 0,Y 587.141,Z 405.2,A -85,B 0,C 180,E1 -1527.943,E2 -1527.943} C_VEL
LIN {X 0,Y 587.14,Z 406.785,A -85,B 0,C 180,E1 -1529.315,E2 -1529.315} C_VEL
LIN {X 0,Y 587.137,Z 407,A -85,B 0,C 180,E1 -1530.001,E2 -1530.001} C_VEL
LIN {X 0,Y 587.147,Z 406.185,A -85,B 0,C 180,E1 -1531.372,E2 -1531.372} C_VEL
LIN {X 0,Y 587.141,Z 405.199,A -85,B 0,C 180,E1 -1532.058,E2 -1532.058} C_VEL
LIN {X 0,Y 587.132,Z 403.808,A -85,B 0,C 180,E1 -1532.745,E2 -1532.745} C_VEL
LIN {X 0,Y 587.213,Z 400.894,A -85,B 0,C 180,E1 -1533.775,E2 -1533.775} C_VEL
LIN {X 0,Y 587.147,Z 396.947,A -85,B 0,C 180,E1 -1534.807,E2 -1534.807} C_VEL
LIN {X 0,Y 587.218,Z 390.874,A -85,B 0,C 180,E1 -1536.012,E2 -1536.012} C_VEL
LIN {X 0,Y 587.245,Z 384.233,A -85,B 0,C 180,E1 -1537.047,E2 -1537.047} C_VEL
LIN {X 0,Y 587.3,Z 375.985,A -85,B 0,C 180,E1 -1538.084,E2 -1538.084} C_VEL
LIN {X 0,Y 587.344,Z 367.532,A -85,B 0,C 180,E1 -1538.95,E2 -1538.95} C_VEL
LIN {X 0,Y 587.419,Z 357.089,A -85,B 0,C 180,E1 -1539.817,E2 -1539.817} C_VEL
LIN {X 0,Y 587.497,Z 346.747,A -85,B 0,C 180,E1 -1540.512,E2 -1540.512} C_VEL
LIN {X 0,Y 587.562,Z 334.807,A -85,B 0,C 180,E1 -1541.149,E2 -1541.149} C_VEL
LIN {X 0,Y 587.63,Z 322.584,A -85,B 0,C 180,E1 -1541.64,E2 -1541.64} C_VEL
LIN {X 0,Y 587.704,Z 309.411,A -85,B 0,C 180,E1 -1542.015,E2 -1542.015} C_VEL
LIN {X 0,Y 587.778,Z 297.043,A -85,B 0,C 180,E1 -1542.232,E2 -1542.232} C_VEL
LIN {X 0,Y 587.703,Z 196.888,A -85,B 0,C 180,E1 -1543.463,E2 -1543.463} C_VEL
LIN {X 0,Y 587.381,Z 194.788,A -85,B 0,C 180,E1 -1543.515,E2 -1543.515} C_VEL
LIN {X 0,Y 587.543,Z 174.797,A -85,B 0,C 180,E1 -1546.326,E2 -1546.326} C_VEL
LIN {X 0,Y 587.672,Z 155.129,A -85,B 0,C 180,E1 -1549.132,E2 -1549.132} C_VEL
LIN {X 0,Y 587.772,Z 135.729,A -85,B 0,C 180,E1 -1551.942,E2 -1551.942} C_VEL
LIN {X 0,Y 587.287,Z 130.358,A -85,B 0,C 180,E1 -1552.732,E2 -1552.732} C_VEL
LIN {X 0,Y 587.297,Z 130.332,A -85,B 0,C 180,E1 -1555.519,E2 -1555.519} C_VEL
LIN {X 0,Y 587.287,Z 130.328,A -85,B 0,C 180,E1 -1557.821,E2 -1557.821} C_VEL
LIN {X 0,Y 587.289,Z 130.325,A -85,B 0,C 180,E1 -1560.501,E2 -1560.501} C_VEL
LIN {X 0,Y 587.289,Z 130.334,A -85,B 0,C 180,E1 -1563.104,E2 -1563.104} C_VEL
LIN {X 0,Y 587.254,Z 130.332,A -85,B 0,C 180,E1 -1565.531,E2 -1565.531} C_VEL
LIN {X 0,Y 587.314,Z 130.322,A -85,B 0,C 180,E1 -1567.835,E2 -1567.835} C_VEL
LIN {X 0,Y 587.293,Z 130.325,A -85,B 0,C 180,E1 -1570.257,E2 -1570.257} C_VEL
LIN {X 0,Y 587.289,Z 130.33,A -85,B 0,C 180,E1 -1573.115,E2 -1573.115} C_VEL
LIN {X 0,Y 587.301,Z 130.323,A -85,B 0,C 180,E1 -1576.047,E2 -1576.047} C_VEL
LIN {X 0,Y 587.31,Z 130.328,A -85,B 0,C 180,E1 -1578.929,E2 -1578.929} C_VEL
LIN {X 0,Y 587.303,Z 130.322,A -85,B 0,C 180,E1 -1581.518,E2 -1581.518} C_VEL
LIN {X 0,Y 587.275,Z 130.328,A -85,B 0,C 180,E1 -1584.099,E2 -1584.099} C_VEL
LIN {X 0,Y 587.334,Z 130.323,A -85,B 0,C 180,E1 -1586.89,E2 -1586.89} C_VEL
LIN {X 0,Y 587.307,Z 130.322,A -85,B 0,C 180,E1 -1589.496,E2 -1589.496} C_VEL
LIN {X 0,Y 587.298,Z 130.332,A -85,B 0,C 180,E1 -1592.318,E2 -1592.318} C_VEL
LIN {X 0,Y 587.304,Z 130.322,A -85,B 0,C 180,E1 -1595.239,E2 -1595.239} C_VEL
LIN {X 0,Y 587.307,Z 130.332,A -85,B 0,C 180,E1 -1598.225,E2 -1598.225} C_VEL
LIN {X 0,Y 587.325,Z 130.32,A -85,B 0,C 180,E1 -1601.15,E2 -1601.15} C_VEL
LIN {X 0,Y 587.296,Z 130.333,A -85,B 0,C 180,E1 -1604.024,E2 -1604.024} C_VEL
LIN {X 0,Y 587.348,Z 130.325,A -85,B 0,C 180,E1 -1606.154,E2 -1606.154} C_VEL
LIN {X 0,Y 587.341,Z 130.318,A -85,B 0,C 180,E1 -1608.963,E2 -1608.963} C_VEL
LIN {X 0,Y 587.338,Z 130.327,A -85,B 0,C 180,E1 -1611.744,E2 -1611.744} C_VEL
LIN {X 0,Y 587.341,Z 130.319,A -85,B 0,C 180,E1 -1614.507,E2 -1614.507} C_VEL
LIN {X 0,Y 587.35,Z 130.32,A -85,B 0,C 180,E1 -1617.257,E2 -1617.257} C_VEL
LIN {X 0,Y 587.384,Z 130.317,A -85,B 0,C 180,E1 -1620,E2 -1620} C_VEL
LIN {X 0,Y 587.349,Z 130.318,A -85,B 0,C 180,E1 -1622.744,E2 -1622.744} C_VEL
LIN {X 0,Y 587.351,Z 130.327,A -85,B 0,C 180,E1 -1625.493,E2 -1625.493} C_VEL
LIN {X 0,Y 587.374,Z 130.475,A -85,B 0,C 180,E1 -1628.472,E2 -1628.472} C_VEL
LIN {X 0,Y 587.479,Z 141.27,A -85,B 0,C 180,E1 -1630.338,E2 -1630.338} C_VEL
LIN {X 0,Y 587.414,Z 156.694,A -85,B 0,C 180,E1 -1632.964,E2 -1632.964} C_VEL
LIN {X 0,Y 587.351,Z 166.127,A -85,B 0,C 180,E1 -1634.553,E2 -1634.553} C_VEL
LIN {X 0,Y 587.881,Z 170.356,A -85,B 0,C 180,E1 -1634.628,E2 -1634.628} C_VEL
LIN {X 0,Y 587.859,Z 174.802,A -85,B 0,C 180,E1 -1634.683,E2 -1634.683} C_VEL
LIN {X 0,Y 587.197,Z 180.646,A -85,B 0,C 180,E1 -1634.739,E2 -1634.739} C_VEL
LIN {X 0,Y 581.596,Z 199.651,A -85,B 0,C 180,E1 -1634.845,E2 -1634.845} C_VEL
LIN {X 0,Y 580.925,Z 205.496,A -85,B 0,C 180,E1 -1634.902,E2 -1634.902} C_VEL
LIN {X 0,Y 580.796,Z 272.848,A -85,B 0,C 180,E1 -1635.754,E2 -1635.754} C_VEL
LIN {X 0,Y 580.712,Z 286.604,A -85,B 0,C 180,E1 -1636.072,E2 -1636.072} C_VEL
LIN {X 0,Y 580.652,Z 298.27,A -85,B 0,C 180,E1 -1636.48,E2 -1636.48} C_VEL
LIN {X 0,Y 580.575,Z 310.316,A -85,B 0,C 180,E1 -1637.037,E2 -1637.037} C_VEL
LIN {X 0,Y 580.441,Z 321.486,A -85,B 0,C 180,E1 -1637.711,E2 -1637.711} C_VEL
LIN {X 0,Y 580.377,Z 331.343,A -85,B 0,C 180,E1 -1638.443,E2 -1638.443} C_VEL
LIN {X 0,Y 580.299,Z 340.263,A -85,B 0,C 180,E1 -1639.252,E2 -1639.252} C_VEL
LIN {X 0,Y 580.193,Z 348.778,A -85,B 0,C 180,E1 -1640.196,E2 -1640.196} C_VEL
LIN {X 0,Y 580.204,Z 355.816,A -85,B 0,C 180,E1 -1641.139,E2 -1641.139} C_VEL
LIN {X 0,Y 580.108,Z 361.456,A -85,B 0,C 180,E1 -1642.06,E2 -1642.06} C_VEL
LIN {X 0,Y 580.109,Z 367.124,A -85,B 0,C 180,E1 -1643.229,E2 -1643.229} C_VEL
LIN {X 0,Y 580.073,Z 371.219,A -85,B 0,C 180,E1 -1644.327,E2 -1644.327} C_VEL
LIN {X 0,Y 580.046,Z 373.356,A -85,B 0,C 180,E1 -1645.092,E2 -1645.092} C_VEL
LIN {X 0,Y 580.048,Z 375.721,A -85,B 0,C 180,E1 -1646.284,E2 -1646.284} C_VEL
LIN {X 0,Y 580.049,Z 376.954,A -85,B 0,C 180,E1 -1647.811,E2 -1647.811} C_VEL
LIN {X 0,Y 580.074,Z 376.347,A -85,B 0,C 180,E1 -1649.269,E2 -1649.269} C_VEL
LIN {X 0,Y 580.072,Z 374.311,A -85,B 0,C 180,E1 -1650.588,E2 -1650.588} C_VEL
LIN {X 0,Y 580.062,Z 372.31,A -85,B 0,C 180,E1 -1651.399,E2 -1651.399} C_VEL
LIN {X 0,Y 580.073,Z 368.109,A -85,B 0,C 180,E1 -1652.626,E2 -1652.626} C_VEL
LIN {X 0,Y 580.118,Z 363.952,A -85,B 0,C 180,E1 -1653.549,E2 -1653.549} C_VEL
LIN {X 0,Y 580.122,Z 357.401,A -85,B 0,C 180,E1 -1654.708,E2 -1654.708} C_VEL
LIN {X 0,Y 580.201,Z 349.102,A -85,B 0,C 180,E1 -1655.855,E2 -1655.855} C_VEL
LIN {X 0,Y 580.274,Z 340.803,A -85,B 0,C 180,E1 -1656.783,E2 -1656.783} C_VEL
LIN {X 0,Y 580.363,Z 330.672,A -85,B 0,C 180,E1 -1657.701,E2 -1657.701} C_VEL
LIN {X 0,Y 580.445,Z 320.194,A -85,B 0,C 180,E1 -1658.466,E2 -1658.466} C_VEL
LIN {X 0,Y 580.544,Z 308.51,A -85,B 0,C 180,E1 -1659.146,E2 -1659.146} C_VEL
LIN {X 0,Y 580.68,Z 296.977,A -85,B 0,C 180,E1 -1659.661,E2 -1659.661} C_VEL
LIN {X 0,Y 580.764,Z 284.352,A -85,B 0,C 180,E1 -1660.083,E2 -1660.083} C_VEL
LIN {X 0,Y 580.797,Z 271.85,A -85,B 0,C 180,E1 -1660.352,E2 -1660.352} C_VEL
LIN {X 0,Y 580.851,Z 169.473,A -85,B 0,C 180,E1 -1661.638,E2 -1661.638} C_VEL
LIN {X 0,Y 580.344,Z 166.124,A -85,B 0,C 180,E1 -1661.703,E2 -1661.703} C_VEL
LIN {X 0,Y 580.455,Z 148.019,A -85,B 0,C 180,E1 -1664.804,E2 -1664.804} C_VEL
LIN {X 0,Y 580.539,Z 133.561,A -85,B 0,C 180,E1 -1667.317,E2 -1667.317} C_VEL
LIN {X 0,Y 580.272,Z 131.203,A -85,B 0,C 180,E1 -1667.767,E2 -1667.767} C_VEL
LIN {X 0,Y 580.284,Z 131.204,A -85,B 0,C 180,E1 -1670.817,E2 -1670.817} C_VEL
LIN {X 0,Y 580.246,Z 131.202,A -85,B 0,C 180,E1 -1673.594,E2 -1673.594} C_VEL
LIN {X 0,Y 580.277,Z 131.202,A -85,B 0,C 180,E1 -1676.142,E2 -1676.142} C_VEL
LIN {X 0,Y 580.265,Z 131.206,A -85,B 0,C 180,E1 -1678.613,E2 -1678.613} C_VEL
LIN {X 0,Y 580.251,Z 131.202,A -85,B 0,C 180,E1 -1681.021,E2 -1681.021} C_VEL
LIN {X 0,Y 580.264,Z 131.2,A -85,B 0,C 180,E1 -1683.673,E2 -1683.673} C_VEL
LIN {X 0,Y 580.249,Z 131.209,A -85,B 0,C 180,E1 -1686.44,E2 -1686.44} C_VEL
LIN {X 0,Y 580.249,Z 131.201,A -85,B 0,C 180,E1 -1689.436,E2 -1689.436} C_VEL
LIN {X 0,Y 580.229,Z 131.206,A -85,B 0,C 180,E1 -1691.643,E2 -1691.643} C_VEL
LIN {X 0,Y 580.268,Z 131.202,A -85,B 0,C 180,E1 -1694.546,E2 -1694.546} C_VEL
LIN {X 0,Y 580.24,Z 131.204,A -85,B 0,C 180,E1 -1696.695,E2 -1696.695} C_VEL
LIN {X 0,Y 580.274,Z 131.198,A -85,B 0,C 180,E1 -1698.826,E2 -1698.826} C_VEL
LIN {X 0,Y 580.298,Z 131.199,A -85,B 0,C 180,E1 -1701.643,E2 -1701.643} C_VEL
LIN {X 0,Y 580.301,Z 131.197,A -85,B 0,C 180,E1 -1704.439,E2 -1704.439} C_VEL
LIN {X 0,Y 580.341,Z 131.199,A -85,B 0,C 180,E1 -1707.917,E2 -1707.917} C_VEL
LIN {X 0,Y 580.352,Z 131.195,A -85,B 0,C 180,E1 -1709.999,E2 -1709.999} C_VEL
LIN {X 0,Y 580.304,Z 131.194,A -85,B 0,C 180,E1 -1712.776,E2 -1712.776} C_VEL
LIN {X 0,Y 580.304,Z 131.202,A -85,B 0,C 180,E1 -1715.559,E2 -1715.559} C_VEL
LIN {X 0,Y 580.295,Z 131.196,A -85,B 0,C 180,E1 -1718.356,E2 -1718.356} C_VEL
LIN {X 0,Y 580.271,Z 131.202,A -85,B 0,C 180,E1 -1721.173,E2 -1721.173} C_VEL
LIN {X 0,Y 580.271,Z 131.199,A -85,B 0,C 180,E1 -1724.319,E2 -1724.319} C_VEL
LIN {X 0,Y 580.253,Z 131.202,A -85,B 0,C 180,E1 -1726.898,E2 -1726.898} C_VEL
LIN {X 0,Y 580.27,Z 131.202,A -85,B 0,C 180,E1 -1729.823,E2 -1729.823} C_VEL
LIN {X 0,Y 580.229,Z 131.204,A -85,B 0,C 180,E1 -1732.054,E2 -1732.054} C_VEL
LIN {X 0,Y 580.274,Z 131.204,A -85,B 0,C 180,E1 -1735.08,E2 -1735.08} C_VEL
LIN {X 0,Y 580.239,Z 131.204,A -85,B 0,C 180,E1 -1737.847,E2 -1737.847} C_VEL
LIN {X 0,Y 580.241,Z 131.205,A -85,B 0,C 180,E1 -1740.686,E2 -1740.686} C_VEL
LIN {X 0,Y 580.275,Z 131.204,A -85,B 0,C 180,E1 -1743.311,E2 -1743.311} C_VEL
LIN {X 0,Y 580.213,Z 131.206,A -85,B 0,C 180,E1 -1745.751,E2 -1745.751} C_VEL
LIN {X 0,Y 580.276,Z 131.198,A -85,B 0,C 180,E1 -1748.146,E2 -1748.146} C_VEL
LIN {X 0,Y 580.272,Z 131.206,A -85,B 0,C 180,E1 -1750.845,E2 -1750.845} C_VEL
LIN {X 0,Y 580.232,Z 131.204,A -85,B 0,C 180,E1 -1753.661,E2 -1753.661} C_VEL
LIN {X 0,Y 580.232,Z 131.205,A -85,B 0,C 180,E1 -1756.337,E2 -1756.337} C_VEL
LIN {X 0,Y 580.251,Z 131.205,A -85,B 0,C 180,E1 -1759.152,E2 -1759.152} C_VEL
LIN {X 0,Y 580.271,Z 131.199,A -85,B 0,C 180,E1 -1761.928,E2 -1761.928} C_VEL
LIN {X 0,Y 580.218,Z 131.211,A -85,B 0,C 180,E1 -1764.45,E2 -1764.45} C_VEL
LIN {X 0,Y 580.275,Z 131.202,A -85,B 0,C 180,E1 -1766.974,E2 -1766.974} C_VEL
LIN {X 0,Y 580.262,Z 131.199,A -85,B 0,C 180,E1 -1769.423,E2 -1769.423} C_VEL
LIN {X 0,Y 580.233,Z 131.207,A -85,B 0,C 180,E1 -1772.152,E2 -1772.152} C_VEL
LIN {X 0,Y 580.273,Z 131.201,A -85,B 0,C 180,E1 -1774.918,E2 -1774.918} C_VEL
LIN {X 0,Y 580.224,Z 131.207,A -85,B 0,C 180,E1 -1777.945,E2 -1777.945} C_VEL
LIN {X 0,Y 580.268,Z 131.2,A -85,B 0,C 180,E1 -1780.912,E2 -1780.912} C_VEL
LIN {X 0,Y 580.229,Z 131.207,A -85,B 0,C 180,E1 -1783.824,E2 -1783.824} C_VEL
LIN {X 0,Y 580.286,Z 131.202,A -85,B 0,C 180,E1 -1785.982,E2 -1785.982} C_VEL
LIN {X 0,Y 580.26,Z 131.201,A -85,B 0,C 180,E1 -1788.826,E2 -1788.826} C_VEL
LIN {X 0,Y 580.286,Z 131.199,A -85,B 0,C 180,E1 -1791.643,E2 -1791.643} C_VEL
LIN {X 0,Y 580.298,Z 131.199,A -85,B 0,C 180,E1 -1794.44,E2 -1794.44} C_VEL
LIN {X 0,Y 580.335,Z 131.199,A -85,B 0,C 180,E1 -1797.918,E2 -1797.918} C_VEL
LIN {X 0,Y 580.341,Z 131.199,A -85,B 0,C 180,E1 -1800,E2 -1800} C_VEL
LIN {X 0,Y 580.293,Z 131.195,A -85,B 0,C 180,E1 -1802.777,E2 -1802.777} C_VEL
LIN {X 0,Y 580.293,Z 131.201,A -85,B 0,C 180,E1 -1805.56,E2 -1805.56} C_VEL
LIN {X 0,Y 580.284,Z 131.198,A -85,B 0,C 180,E1 -1808.357,E2 -1808.357} C_VEL
LIN {X 0,Y 580.259,Z 131.202,A -85,B 0,C 180,E1 -1811.174,E2 -1811.174} C_VEL
LIN {X 0,Y 580.283,Z 131.201,A -85,B 0,C 180,E1 -1814.018,E2 -1814.018} C_VEL
LIN {X 0,Y 580.242,Z 131.203,A -85,B 0,C 180,E1 -1816.899,E2 -1816.899} C_VEL
LIN {X 0,Y 580.26,Z 131.205,A -85,B 0,C 180,E1 -1819.824,E2 -1819.824} C_VEL
LIN {X 0,Y 580.219,Z 131.207,A -85,B 0,C 180,E1 -1822.055,E2 -1822.055} C_VEL
LIN {X 0,Y 580.241,Z 131.203,A -85,B 0,C 180,E1 -1824.715,E2 -1824.715} C_VEL
LIN {X 0,Y 580.236,Z 131.212,A -85,B 0,C 180,E1 -1827.404,E2 -1827.404} C_VEL
LIN {X 0,Y 580.238,Z 131.205,A -85,B 0,C 180,E1 -1829.776,E2 -1829.776} C_VEL
LIN {X 0,Y 580.274,Z 131.198,A -85,B 0,C 180,E1 -1832.202,E2 -1832.202} C_VEL
LIN {X 0,Y 580.261,Z 131.202,A -85,B 0,C 180,E1 -1834.698,E2 -1834.698} C_VEL
LIN {X 0,Y 580.272,Z 131.206,A -85,B 0,C 180,E1 -1837.27,E2 -1837.27} C_VEL
LIN {X 0,Y 580.265,Z 131.199,A -85,B 0,C 180,E1 -1840.269,E2 -1840.269} C_VEL
LIN {X 0,Y 580.24,Z 131.207,A -85,B 0,C 180,E1 -1842.71,E2 -1842.71} C_VEL
LIN {X 0,Y 580.244,Z 131.203,A -85,B 0,C 180,E1 -1845.612,E2 -1845.612} C_VEL
LIN {X 0,Y 580.23,Z 131.204,A -85,B 0,C 180,E1 -1848.228,E2 -1848.228} C_VEL
LIN {X 0,Y 580.253,Z 131.209,A -85,B 0,C 180,E1 -1850.964,E2 -1850.964} C_VEL
LIN {X 0,Y 580.226,Z 131.204,A -85,B 0,C 180,E1 -1853.594,E2 -1853.594} C_VEL
LIN {X 0,Y 580.258,Z 131.201,A -85,B 0,C 180,E1 -1856.142,E2 -1856.142} C_VEL
LIN {X 0,Y 580.234,Z 131.211,A -85,B 0,C 180,E1 -1858.613,E2 -1858.613} C_VEL
LIN {X 0,Y 580.239,Z 131.207,A -85,B 0,C 180,E1 -1861.022,E2 -1861.022} C_VEL
LIN {X 0,Y 580.246,Z 131.202,A -85,B 0,C 180,E1 -1863.676,E2 -1863.676} C_VEL
LIN {X 0,Y 580.236,Z 131.212,A -85,B 0,C 180,E1 -1866.441,E2 -1866.441} C_VEL
LIN {X 0,Y 580.226,Z 131.233,A -85,B 0,C 180,E1 -1867.113,E2 -1867.113} C_VEL
LIN {X 0,Y 580.833,Z 135.62,A -85,B 0,C 180,E1 -1867.783,E2 -1867.783} C_VEL
LIN {X 0,Y 580.708,Z 154.388,A -85,B 0,C 180,E1 -1870.522,E2 -1870.522} C_VEL
LIN {X 0,Y 580.536,Z 173.546,A -85,B 0,C 180,E1 -1873.291,E2 -1873.291} C_VEL
LIN {X 0,Y 580.4,Z 194.64,A -85,B 0,C 180,E1 -1876.298,E2 -1876.298} C_VEL
LIN {X 0,Y 580.417,Z 195.196,A -85,B 0,C 180,E1 -1876.343,E2 -1876.343} C_VEL
LIN {X 0,Y 580.949,Z 200.562,A -85,B 0,C 180,E1 -1876.423,E2 -1876.423} C_VEL
LIN {X 0,Y 580.81,Z 302.98,A -85,B 0,C 180,E1 -1877.709,E2 -1877.709} C_VEL
LIN {X 0,Y 580.726,Z 316.241,A -85,B 0,C 180,E1 -1878.017,E2 -1878.017} C_VEL
LIN {X 0,Y 580.645,Z 328.392,A -85,B 0,C 180,E1 -1878.437,E2 -1878.437} C_VEL
LIN {X 0,Y 580.542,Z 340.639,A -85,B 0,C 180,E1 -1879.009,E2 -1879.009} C_VEL
LIN {X 0,Y 580.44,Z 352.21,A -85,B 0,C 180,E1 -1879.713,E2 -1879.713} C_VEL
LIN {X 0,Y 580.345,Z 362.609,A -85,B 0,C 180,E1 -1880.503,E2 -1880.503} C_VEL
LIN {X 0,Y 580.271,Z 371.119,A -85,B 0,C 180,E1 -1881.293,E2 -1881.293} C_VEL
LIN {X 0,Y 580.221,Z 378.966,A -85,B 0,C 180,E1 -1882.169,E2 -1882.169} C_VEL
LIN {X 0,Y 580.153,Z 386.654,A -85,B 0,C 180,E1 -1883.222,E2 -1883.222} C_VEL
LIN {X 0,Y 580.139,Z 393.683,A -85,B 0,C 180,E1 -1884.439,E2 -1884.439} C_VEL
LIN {X 0,Y 580.108,Z 398.375,A -85,B 0,C 180,E1 -1885.484,E2 -1885.484} C_VEL
LIN {X 0,Y 580.122,Z 401.959,A -85,B 0,C 180,E1 -1886.528,E2 -1886.528} C_VEL
LIN {X 0,Y 580.043,Z 403.81,A -85,B 0,C 180,E1 -1887.223,E2 -1887.223} C_VEL
LIN {X 0,Y 580.04,Z 405.199,A -85,B 0,C 180,E1 -1887.917,E2 -1887.917} C_VEL
LIN {X 0,Y 580.04,Z 406.785,A -85,B 0,C 180,E1 -1889.306,E2 -1889.306} C_VEL
LIN {X 0,Y 580.037,Z 407,A -85,B 0,C 180,E1 -1890.001,E2 -1890.001} C_VEL
LIN {X 0,Y 580.047,Z 406.186,A -85,B 0,C 180,E1 -1891.389,E2 -1891.389} C_VEL
LIN {X 0,Y 580.04,Z 405.198,A -85,B 0,C 180,E1 -1892.084,E2 -1892.084} C_VEL
LIN {X 0,Y 580.043,Z 403.808,A -85,B 0,C 180,E1 -1892.779,E2 -1892.779} C_VEL
LIN {X 0,Y 580.11,Z 400.894,A -85,B 0,C 180,E1 -1893.821,E2 -1893.821} C_VEL
LIN {X 0,Y 580.053,Z 396.947,A -85,B 0,C 180,E1 -1894.866,E2 -1894.866} C_VEL
LIN {X 0,Y 580.139,Z 390.873,A -85,B 0,C 180,E1 -1896.085,E2 -1896.085} C_VEL
LIN {X 0,Y 580.185,Z 384.233,A -85,B 0,C 180,E1 -1897.133,E2 -1897.133} C_VEL
LIN {X 0,Y 580.251,Z 375.986,A -85,B 0,C 180,E1 -1898.182,E2 -1898.182} C_VEL
LIN {X 0,Y 580.308,Z 367.532,A -85,B 0,C 180,E1 -1899.059,E2 -1899.059} C_VEL
LIN {X 0,Y 580.422,Z 357.09,A -85,B 0,C 180,E1 -1899.936,E2 -1899.936} C_VEL
LIN {X 0,Y 580.507,Z 346.745,A -85,B 0,C 180,E1 -1900.64,E2 -1900.64} C_VEL
LIN {X 0,Y 580.597,Z 335.237,A -85,B 0,C 180,E1 -1901.264,E2 -1901.264} C_VEL
LIN {X 0,Y 580.683,Z 322.455,A -85,B 0,C 180,E1 -1901.785,E2 -1901.785} C_VEL
LIN {X 0,Y 580.756,Z 309.41,A -85,B 0,C 180,E1 -1902.16,E2 -1902.16} C_VEL
LIN {X 0,Y 580.854,Z 297.043,A -85,B 0,C 180,E1 -1902.38,E2 -1902.38} C_VEL
LIN {X 0,Y 580.787,Z 197.558,A -85,B 0,C 180,E1 -1903.618,E2 -1903.618} C_VEL
LIN {X 0,Y 580.386,Z 194.788,A -85,B 0,C 180,E1 -1903.681,E2 -1903.681} C_VEL
LIN {X 0,Y 580.538,Z 174.797,A -85,B 0,C 180,E1 -1906.529,E2 -1906.529} C_VEL
LIN {X 0,Y 580.703,Z 155.853,A -85,B 0,C 180,E1 -1909.265,E2 -1909.265} C_VEL
LIN {X 0,Y 580.849,Z 138.023,A -85,B 0,C 180,E1 -1911.843,E2 -1911.843} C_VEL
LIN {X 0,Y 580.521,Z 132.849,A -85,B 0,C 180,E1 -1912.606,E2 -1912.606} C_VEL
LIN {X 0,Y 580.249,Z 131.209,A -85,B 0,C 180,E1 -1912.86,E2 -1912.86} C_VEL
LIN {X 0,Y 580.243,Z 131.206,A -85,B 0,C 180,E1 -1915.852,E2 -1915.852} C_VEL
LIN {X 0,Y 580.226,Z 131.205,A -85,B 0,C 180,E1 -1918.19,E2 -1918.19} C_VEL
LIN {X 0,Y 580.242,Z 131.205,A -85,B 0,C 180,E1 -1920.687,E2 -1920.687} C_VEL
LIN {X 0,Y 580.271,Z 131.206,A -85,B 0,C 180,E1 -1923.311,E2 -1923.311} C_VEL
LIN {X 0,Y 580.208,Z 131.208,A -85,B 0,C 180,E1 -1925.751,E2 -1925.751} C_VEL
LIN {X 0,Y 580.275,Z 131.198,A -85,B 0,C 180,E1 -1928.148,E2 -1928.148} C_VEL
LIN {X 0,Y 580.275,Z 131.206,A -85,B 0,C 180,E1 -1930.846,E2 -1930.846} C_VEL
LIN {X 0,Y 580.237,Z 131.203,A -85,B 0,C 180,E1 -1933.662,E2 -1933.662} C_VEL
LIN {X 0,Y 580.238,Z 131.205,A -85,B 0,C 180,E1 -1936.338,E2 -1936.338} C_VEL
LIN {X 0,Y 580.257,Z 131.203,A -85,B 0,C 180,E1 -1939.153,E2 -1939.153} C_VEL
LIN {X 0,Y 580.278,Z 131.198,A -85,B 0,C 180,E1 -1941.929,E2 -1941.929} C_VEL
LIN {X 0,Y 580.226,Z 131.211,A -85,B 0,C 180,E1 -1944.451,E2 -1944.451} C_VEL
LIN {X 0,Y 580.284,Z 131.2,A -85,B 0,C 180,E1 -1946.975,E2 -1946.975} C_VEL
LIN {X 0,Y 580.271,Z 131.198,A -85,B 0,C 180,E1 -1949.424,E2 -1949.424} C_VEL
LIN {X 0,Y 580.243,Z 131.208,A -85,B 0,C 180,E1 -1952.153,E2 -1952.153} C_VEL
LIN {X 0,Y 580.284,Z 131.198,A -85,B 0,C 180,E1 -1954.919,E2 -1954.919} C_VEL
LIN {X 0,Y 580.251,Z 131.206,A -85,B 0,C 180,E1 -1957.947,E2 -1957.947} C_VEL
LIN {X 0,Y 580.28,Z 131.198,A -85,B 0,C 180,E1 -1960.913,E2 -1960.913} C_VEL
LIN {X 0,Y 580.243,Z 131.208,A -85,B 0,C 180,E1 -1963.825,E2 -1963.825} C_VEL
LIN {X 0,Y 580.306,Z 131.204,A -85,B 0,C 180,E1 -1965.983,E2 -1965.983} C_VEL
LIN {X 0,Y 580.31,Z 131.194,A -85,B 0,C 180,E1 -1968.827,E2 -1968.827} C_VEL
LIN {X 0,Y 580.306,Z 131.201,A -85,B 0,C 180,E1 -1971.644,E2 -1971.644} C_VEL
LIN {X 0,Y 580.31,Z 131.195,A -85,B 0,C 180,E1 -1974.44,E2 -1974.44} C_VEL
LIN {X 0,Y 580.343,Z 131.196,A -85,B 0,C 180,E1 -1977.918,E2 -1977.918} C_VEL
LIN {X 0,Y 580.353,Z 131.193,A -85,B 0,C 180,E1 -1980,E2 -1980} C_VEL
LIN {X 0,Y 580.318,Z 131.194,A -85,B 0,C 180,E1 -1982.777,E2 -1982.777} C_VEL
LIN {X 0,Y 580.317,Z 131.203,A -85,B 0,C 180,E1 -1985.56,E2 -1985.56} C_VEL
LIN {X 0,Y 580.32,Z 131.393,A -85,B 0,C 180,E1 -1988.4,E2 -1988.4} C_VEL
LIN {X 0,Y 580.491,Z 140.222,A -85,B 0,C 180,E1 -1989.935,E2 -1989.935} C_VEL
LIN {X 0,Y 580.403,Z 156.636,A -85,B 0,C 180,E1 -1992.767,E2 -1992.767} C_VEL
LIN {X 0,Y 580.319,Z 166.081,A -85,B 0,C 180,E1 -1994.379,E2 -1994.379} C_VEL
LIN {X 0,Y 580.985,Z 170.936,A -85,B 0,C 180,E1 -1994.473,E2 -1994.473} C_VEL
LIN {X 0,Y 580.925,Z 205.496,A -85,B 0,C 180,E1 -1994.902,E2 -1994.902} C_VEL
LIN {X 0,Y 580.242,Z 211.34,A -85,B 0,C 180,E1 -1994.959,E2 -1994.959} C_VEL
LIN {X 0,Y 574.593,Z 230.33,A -85,B 0,C 180,E1 -1995.067,E2 -1995.067} C_VEL
LIN {X 0,Y 573.971,Z 236.172,A -85,B 0,C 180,E1 -1995.126,E2 -1995.126} C_VEL
LIN {X 0,Y 573.869,Z 273.045,A -85,B 0,C 180,E1 -1995.608,E2 -1995.608} C_VEL
LIN {X 0,Y 573.758,Z 286.736,A -85,B 0,C 180,E1 -1995.93,E2 -1995.93} C_VEL
LIN {X 0,Y 573.675,Z 298.964,A -85,B 0,C 180,E1 -1996.366,E2 -1996.366} C_VEL
LIN {X 0,Y 573.586,Z 310.526,A -85,B 0,C 180,E1 -1996.912,E2 -1996.912} C_VEL
LIN {X 0,Y 573.448,Z 321.212,A -85,B 0,C 180,E1 -1997.566,E2 -1997.566} C_VEL
LIN {X 0,Y 573.362,Z 331.123,A -85,B 0,C 180,E1 -1998.307,E2 -1998.307} C_VEL
LIN {X 0,Y 573.245,Z 341.371,A -85,B 0,C 180,E1 -1999.261,E2 -1999.261} C_VEL
LIN {X 0,Y 573.139,Z 348.624,A -85,B 0,C 180,E1 -2000.081,E2 -2000.081} C_VEL
LIN {X 0,Y 573.112,Z 355.73,A -85,B 0,C 180,E1 -2001.042,E2 -2001.042} C_VEL
LIN {X 0,Y 573.044,Z 361.353,A -85,B 0,C 180,E1 -2001.967,E2 -2001.967} C_VEL
LIN {X 0,Y 573.019,Z 366.864,A -85,B 0,C 180,E1 -2003.109,E2 -2003.109} C_VEL
LIN {X 0,Y 572.997,Z 371.147,A -85,B 0,C 180,E1 -2004.261,E2 -2004.261} C_VEL
LIN {X 0,Y 572.954,Z 374.222,A -85,B 0,C 180,E1 -2005.425,E2 -2005.425} C_VEL
LIN {X 0,Y 572.958,Z 375.937,A -85,B 0,C 180,E1 -2006.435,E2 -2006.435} C_VEL
LIN {X 0,Y 572.954,Z 376.946,A -85,B 0,C 180,E1 -2007.783,E2 -2007.783} C_VEL
LIN {X 0,Y 572.937,Z 376.846,A -85,B 0,C 180,E1 -2008.581,E2 -2008.581} C_VEL
LIN {X 0,Y 572.976,Z 376.172,A -85,B 0,C 180,E1 -2009.439,E2 -2009.439} C_VEL
LIN {X 0,Y 572.982,Z 373.841,A -85,B 0,C 180,E1 -2010.84,E2 -2010.84} C_VEL
LIN {X 0,Y 572.99,Z 369.945,A -85,B 0,C 180,E1 -2012.186,E2 -2012.186} C_VEL
LIN {X 0,Y 573.038,Z 364.55,A -85,B 0,C 180,E1 -2013.498,E2 -2013.498} C_VEL
LIN {X 0,Y 573.045,Z 358.88,A -85,B 0,C 180,E1 -2014.545,E2 -2014.545} C_VEL
LIN {X 0,Y 573.131,Z 351.671,A -85,B 0,C 180,E1 -2015.625,E2 -2015.625} C_VEL
LIN {X 0,Y 573.191,Z 343.549,A -85,B 0,C 180,E1 -2016.599,E2 -2016.599} C_VEL
LIN {X 0,Y 573.318,Z 334.903,A -85,B 0,C 180,E1 -2017.453,E2 -2017.453} C_VEL
LIN {X 0,Y 573.392,Z 324.046,A -85,B 0,C 180,E1 -2018.33,E2 -2018.33} C_VEL
LIN {X 0,Y 573.498,Z 313.286,A -85,B 0,C 180,E1 -2019.02,E2 -2019.02} C_VEL
LIN {X 0,Y 573.666,Z 301.277,A -85,B 0,C 180,E1 -2019.63,E2 -2019.63} C_VEL
LIN {X 0,Y 573.765,Z 288.835,A -85,B 0,C 180,E1 -2020.093,E2 -2020.093} C_VEL
LIN {X 0,Y 573.852,Z 275.972,A -85,B 0,C 180,E1 -2020.431,E2 -2020.431} C_VEL
LIN {X 0,Y 573.915,Z 255.842,A -85,B 0,C 180,E1 -2020.718,E2 -2020.718} C_VEL
LIN {X 0,Y 574.018,Z 170.672,A -85,B 0,C 180,E1 -2021.788,E2 -2021.788} C_VEL
LIN {X 0,Y 573.279,Z 166.176,A -85,B 0,C 180,E1 -2021.866,E2 -2021.866} C_VEL
LIN {X 0,Y 573.425,Z 149.856,A -85,B 0,C 180,E1 -2024.695,E2 -2024.695} C_VEL
LIN {X 0,Y 573.568,Z 134.928,A -85,B 0,C 180,E1 -2027.324,E2 -2027.324} C_VEL
LIN {X 0,Y 573.234,Z 132.081,A -85,B 0,C 180,E1 -2027.872,E2 -2027.872} C_VEL
LIN {X 0,Y 573.237,Z 132.084,A -85,B 0,C 180,E1 -2030.57,E2 -2030.57} C_VEL
LIN {X 0,Y 573.234,Z 132.078,A -85,B 0,C 180,E1 -2033.076,E2 -2033.076} C_VEL
LIN {X 0,Y 573.251,Z 132.073,A -85,B 0,C 180,E1 -2035.67,E2 -2035.67} C_VEL
LIN {X 0,Y 573.229,Z 132.081,A -85,B 0,C 180,E1 -2038.183,E2 -2038.183} C_VEL
LIN {X 0,Y 573.222,Z 132.083,A -85,B 0,C 180,E1 -2040.631,E2 -2040.631} C_VEL
LIN {X 0,Y 573.208,Z 132.078,A -85,B 0,C 180,E1 -2043.515,E2 -2043.515} C_VEL
LIN {X 0,Y 573.198,Z 132.086,A -85,B 0,C 180,E1 -2046.133,E2 -2046.133} C_VEL
LIN {X 0,Y 573.224,Z 132.076,A -85,B 0,C 180,E1 -2049.172,E2 -2049.172} C_VEL
LIN {X 0,Y 573.187,Z 132.081,A -85,B 0,C 180,E1 -2051.41,E2 -2051.41} C_VEL
LIN {X 0,Y 573.207,Z 132.085,A -85,B 0,C 180,E1 -2054.351,E2 -2054.351} C_VEL
LIN {X 0,Y 573.203,Z 132.082,A -85,B 0,C 180,E1 -2056.528,E2 -2056.528} C_VEL
LIN {X 0,Y 573.245,Z 132.075,A -85,B 0,C 180,E1 -2059.402,E2 -2059.402} C_VEL
LIN {X 0,Y 573.224,Z 132.081,A -85,B 0,C 180,E1 -2062.249,E2 -2062.249} C_VEL
LIN {X 0,Y 573.277,Z 132.07,A -85,B 0,C 180,E1 -2065.077,E2 -2065.077} C_VEL
LIN {X 0,Y 573.311,Z 132.075,A -85,B 0,C 180,E1 -2067.892,E2 -2067.892} C_VEL
LIN {X 0,Y 573.32,Z 132.071,A -85,B 0,C 180,E1 -2069.999,E2 -2069.999} C_VEL
LIN {X 0,Y 573.273,Z 132.07,A -85,B 0,C 180,E1 -2072.81,E2 -2072.81} C_VEL
LIN {X 0,Y 573.272,Z 132.079,A -85,B 0,C 180,E1 -2075.628,E2 -2075.628} C_VEL
LIN {X 0,Y 573.236,Z 132.075,A -85,B 0,C 180,E1 -2078.46,E2 -2078.46} C_VEL
LIN {X 0,Y 573.239,Z 132.08,A -85,B 0,C 180,E1 -2081.312,E2 -2081.312} C_VEL
LIN {X 0,Y 573.229,Z 132.075,A -85,B 0,C 180,E1 -2084.401,E2 -2084.401} C_VEL
LIN {X 0,Y 573.195,Z 132.084,A -85,B 0,C 180,E1 -2087.113,E2 -2087.113} C_VEL
LIN {X 0,Y 573.205,Z 132.079,A -85,B 0,C 180,E1 -2090.078,E2 -2090.078} C_VEL
LIN {X 0,Y 573.196,Z 132.08,A -85,B 0,C 180,E1 -2092.339,E2 -2092.339} C_VEL
LIN {X 0,Y 573.221,Z 132.084,A -85,B 0,C 180,E1 -2095.411,E2 -2095.411} C_VEL
LIN {X 0,Y 573.195,Z 132.08,A -85,B 0,C 180,E1 -2098.017,E2 -2098.017} C_VEL
LIN {X 0,Y 573.203,Z 132.084,A -85,B 0,C 180,E1 -2100.877,E2 -2100.877} C_VEL
LIN {X 0,Y 573.241,Z 132.078,A -85,B 0,C 180,E1 -2103.52,E2 -2103.52} C_VEL
LIN {X 0,Y 573.181,Z 132.081,A -85,B 0,C 180,E1 -2106.053,E2 -2106.053} C_VEL
LIN {X 0,Y 573.229,Z 132.08,A -85,B 0,C 180,E1 -2108.702,E2 -2108.702} C_VEL
LIN {X 0,Y 573.197,Z 132.082,A -85,B 0,C 180,E1 -2111.459,E2 -2111.459} C_VEL
LIN {X 0,Y 573.213,Z 132.079,A -85,B 0,C 180,E1 -2114.335,E2 -2114.335} C_VEL
LIN {X 0,Y 573.209,Z 132.08,A -85,B 0,C 180,E1 -2117.361,E2 -2117.361} C_VEL
LIN {X 0,Y 573.223,Z 132.08,A -85,B 0,C 180,E1 -2120.39,E2 -2120.39} C_VEL
LIN {X 0,Y 573.224,Z 132.08,A -85,B 0,C 180,E1 -2123.075,E2 -2123.075} C_VEL
LIN {X 0,Y 573.237,Z 132.074,A -85,B 0,C 180,E1 -2125.669,E2 -2125.669} C_VEL
LIN {X 0,Y 573.218,Z 132.08,A -85,B 0,C 180,E1 -2128.183,E2 -2128.183} C_VEL
LIN {X 0,Y 573.21,Z 132.087,A -85,B 0,C 180,E1 -2130.631,E2 -2130.631} C_VEL
LIN {X 0,Y 573.198,Z 132.079,A -85,B 0,C 180,E1 -2133.514,E2 -2133.514} C_VEL
LIN {X 0,Y 573.186,Z 132.086,A -85,B 0,C 180,E1 -2136.132,E2 -2136.132} C_VEL
LIN {X 0,Y 573.219,Z 132.077,A -85,B 0,C 180,E1 -2139.172,E2 -2139.172} C_VEL
LIN {X 0,Y 573.185,Z 132.081,A -85,B 0,C 180,E1 -2141.41,E2 -2141.41} C_VEL
LIN {X 0,Y 573.196,Z 132.088,A -85,B 0,C 180,E1 -2144.351,E2 -2144.351} C_VEL
LIN {X 0,Y 573.187,Z 132.086,A -85,B 0,C 180,E1 -2146.528,E2 -2146.528} C_VEL
LIN {X 0,Y 573.234,Z 132.075,A -85,B 0,C 180,E1 -2149.403,E2 -2149.403} C_VEL
LIN {X 0,Y 573.211,Z 132.085,A -85,B 0,C 180,E1 -2152.249,E2 -2152.249} C_VEL
LIN {X 0,Y 573.267,Z 132.071,A -85,B 0,C 180,E1 -2155.077,E2 -2155.077} C_VEL
LIN {X 0,Y 573.304,Z 132.075,A -85,B 0,C 180,E1 -2157.892,E2 -2157.892} C_VEL
LIN {X 0,Y 573.31,Z 132.075,A -85,B 0,C 180,E1 -2160,E2 -2160} C_VEL
LIN {X 0,Y 573.261,Z 132.071,A -85,B 0,C 180,E1 -2162.811,E2 -2162.811} C_VEL
LIN {X 0,Y 573.262,Z 132.078,A -85,B 0,C 180,E1 -2165.628,E2 -2165.628} C_VEL
LIN {X 0,Y 573.225,Z 132.077,A -85,B 0,C 180,E1 -2168.46,E2 -2168.46} C_VEL
LIN {X 0,Y 573.227,Z 132.079,A -85,B 0,C 180,E1 -2171.313,E2 -2171.313} C_VEL
LIN {X 0,Y 573.227,Z 132.076,A -85,B 0,C 180,E1 -2174.406,E2 -2174.406} C_VEL
LIN {X 0,Y 573.183,Z 132.084,A -85,B 0,C 180,E1 -2177.114,E2 -2177.114} C_VEL
LIN {X 0,Y 573.195,Z 132.082,A -85,B 0,C 180,E1 -2180.079,E2 -2180.079} C_VEL
LIN {X 0,Y 573.186,Z 132.081,A -85,B 0,C 180,E1 -2182.34,E2 -2182.34} C_VEL
LIN {X 0,Y 573.201,Z 132.089,A -85,B 0,C 180,E1 -2185.413,E2 -2185.413} C_VEL
LIN {X 0,Y 573.185,Z 132.082,A -85,B 0,C 180,E1 -2188.018,E2 -2188.018} C_VEL
LIN {X 0,Y 573.195,Z 132.083,A -85,B 0,C 180,E1 -2190.878,E2 -2190.878} C_VEL
LIN {X 0,Y 573.235,Z 132.08,A -85,B 0,C 180,E1 -2193.521,E2 -2193.521} C_VEL
LIN {X 0,Y 573.173,Z 132.082,A -85,B 0,C 180,E1 -2196.055,E2 -2196.055} C_VEL
LIN {X 0,Y 573.22,Z 132.08,A -85,B 0,C 180,E1 -2198.703,E2 -2198.703} C_VEL
LIN {X 0,Y 573.188,Z 132.083,A -85,B 0,C 180,E1 -2201.589,E2 -2201.589} C_VEL
LIN {X 0,Y 573.202,Z 132.083,A -85,B 0,C 180,E1 -2204.674,E2 -2204.674} C_VEL
LIN {X 0,Y 573.195,Z 132.081,A -85,B 0,C 180,E1 -2207.597,E2 -2207.597} C_VEL
LIN {X 0,Y 573.225,Z 132.081,A -85,B 0,C 180,E1 -2210.571,E2 -2210.571} C_VEL
LIN {X 0,Y 573.22,Z 132.083,A -85,B 0,C 180,E1 -2213.076,E2 -2213.076} C_VEL
LIN {X 0,Y 573.235,Z 132.075,A -85,B 0,C 180,E1 -2215.67,E2 -2215.67} C_VEL
LIN {X 0,Y 573.21,Z 132.08,A -85,B 0,C 180,E1 -2218.184,E2 -2218.184} C_VEL
LIN {X 0,Y 573.21,Z 132.087,A -85,B 0,C 180,E1 -2220.632,E2 -2220.632} C_VEL
LIN {X 0,Y 573.191,Z 132.082,A -85,B 0,C 180,E1 -2223.517,E2 -2223.517} C_VEL
LIN {X 0,Y 573.187,Z 132.086,A -85,B 0,C 180,E1 -2226.133,E2 -2226.133} C_VEL
LIN {X 0,Y 573.218,Z 132.22,A -85,B 0,C 180,E1 -2226.984,E2 -2226.984} C_VEL
LIN {X 0,Y 573.891,Z 136.762,A -85,B 0,C 180,E1 -2227.69,E2 -2227.69} C_VEL
LIN {X 0,Y 573.752,Z 154.556,A -85,B 0,C 180,E1 -2230.316,E2 -2230.316} C_VEL
LIN {X 0,Y 573.541,Z 173.144,A -85,B 0,C 180,E1 -2233.023,E2 -2233.023} C_VEL
LIN {X 0,Y 573.404,Z 193.695,A -85,B 0,C 180,E1 -2235.992,E2 -2235.992} C_VEL
LIN {X 0,Y 573.423,Z 195.196,A -85,B 0,C 180,E1 -2236.173,E2 -2236.173} C_VEL
LIN {X 0,Y 574.06,Z 200.562,A -85,B 0,C 180,E1 -2236.257,E2 -2236.257} C_VEL
LIN {X 0,Y 573.886,Z 302.98,A -85,B 0,C 180,E1 -2237.558,E2 -2237.558} C_VEL
LIN {X 0,Y 573.777,Z 316.241,A -85,B 0,C 180,E1 -2237.87,E2 -2237.87} C_VEL
LIN {X 0,Y 573.697,Z 328.393,A -85,B 0,C 180,E1 -2238.295,E2 -2238.295} C_VEL
LIN {X 0,Y 573.588,Z 339.604,A -85,B 0,C 180,E1 -2238.818,E2 -2238.818} C_VEL
LIN {X 0,Y 573.456,Z 350.916,A -85,B 0,C 180,E1 -2239.497,E2 -2239.497} C_VEL
LIN {X 0,Y 573.35,Z 361.547,A -85,B 0,C 180,E1 -2240.297,E2 -2240.297} C_VEL
LIN {X 0,Y 573.24,Z 371.119,A -85,B 0,C 180,E1 -2241.185,E2 -2241.185} C_VEL
LIN {X 0,Y 573.16,Z 378.966,A -85,B 0,C 180,E1 -2242.072,E2 -2242.072} C_VEL
LIN {X 0,Y 573.072,Z 386.958,A -85,B 0,C 180,E1 -2243.186,E2 -2243.186} C_VEL
LIN {X 0,Y 573.07,Z 393.683,A -85,B 0,C 180,E1 -2244.37,E2 -2244.37} C_VEL
LIN {X 0,Y 573.028,Z 398.375,A -85,B 0,C 180,E1 -2245.428,E2 -2245.428} C_VEL
LIN {X 0,Y 573.022,Z 401.96,A -85,B 0,C 180,E1 -2246.485,E2 -2246.485} C_VEL
LIN {X 0,Y 572.959,Z 403.809,A -85,B 0,C 180,E1 -2247.188,E2 -2247.188} C_VEL
LIN {X 0,Y 572.946,Z 406.186,A -85,B 0,C 180,E1 -2248.595,E2 -2248.595} C_VEL
LIN {X 0,Y 572.938,Z 407,A -85,B 0,C 180,E1 -2250.001,E2 -2250.001} C_VEL
LIN {X 0,Y 572.946,Z 406.185,A -85,B 0,C 180,E1 -2251.406,E2 -2251.406} C_VEL
LIN {X 0,Y 572.94,Z 405.198,A -85,B 0,C 180,E1 -2252.11,E2 -2252.11} C_VEL
LIN {X 0,Y 572.959,Z 403.809,A -85,B 0,C 180,E1 -2252.813,E2 -2252.813} C_VEL
LIN {X 0,Y 573.015,Z 400.894,A -85,B 0,C 180,E1 -2253.869,E2 -2253.869} C_VEL
LIN {X 0,Y 572.963,Z 396.946,A -85,B 0,C 180,E1 -2254.926,E2 -2254.926} C_VEL
LIN {X 0,Y 573.065,Z 390.873,A -85,B 0,C 180,E1 -2256.161,E2 -2256.161} C_VEL
LIN {X 0,Y 573.12,Z 384.233,A -85,B 0,C 180,E1 -2257.221,E2 -2257.221} C_VEL
LIN {X 0,Y 573.201,Z 375.986,A -85,B 0,C 180,E1 -2258.284,E2 -2258.284} C_VEL
LIN {X 0,Y 573.287,Z 367.533,A -85,B 0,C 180,E1 -2259.171,E2 -2259.171} C_VEL
LIN {X 0,Y 573.427,Z 357.088,A -85,B 0,C 180,E1 -2260.059,E2 -2260.059} C_VEL
LIN {X 0,Y 573.544,Z 345.423,A -85,B 0,C 180,E1 -2260.853,E2 -2260.853} C_VEL
LIN {X 0,Y 573.652,Z 334.297,A -85,B 0,C 180,E1 -2261.447,E2 -2261.447} C_VEL
LIN {X 0,Y 573.759,Z 321.153,A -85,B 0,C 180,E1 -2261.975,E2 -2261.975} C_VEL
LIN {X 0,Y 573.856,Z 308.494,A -85,B 0,C 180,E1 -2262.331,E2 -2262.331} C_VEL
LIN {X 0,Y 573.932,Z 295.264,A -85,B 0,C 180,E1 -2262.554,E2 -2262.554} C_VEL
LIN {X 0,Y 573.942,Z 198.675,A -85,B 0,C 180,E1 -2263.77,E2 -2263.77} C_VEL
LIN {X 0,Y 573.388,Z 194.788,A -85,B 0,C 180,E1 -2263.851,E2 -2263.851} C_VEL
LIN {X 0,Y 573.537,Z 174.895,A -85,B 0,C 180,E1 -2266.722,E2 -2266.722} C_VEL
LIN {X 0,Y 573.725,Z 156.422,A -85,B 0,C 180,E1 -2269.398,E2 -2269.398} C_VEL
LIN {X 0,Y 573.862,Z 137.731,A -85,B 0,C 180,E1 -2272.123,E2 -2272.123} C_VEL
LIN {X 0,Y 573.203,Z 132.087,A -85,B 0,C 180,E1 -2272.982,E2 -2272.982} C_VEL
LIN {X 0,Y 573.203,Z 132.089,A -85,B 0,C 180,E1 -2275.413,E2 -2275.413} C_VEL
LIN {X 0,Y 573.195,Z 132.082,A -85,B 0,C 180,E1 -2278.018,E2 -2278.018} C_VEL
LIN {X 0,Y 573.204,Z 132.084,A -85,B 0,C 180,E1 -2280.878,E2 -2280.878} C_VEL
LIN {X 0,Y 573.245,Z 132.078,A -85,B 0,C 180,E1 -2283.521,E2 -2283.521} C_VEL
